ks	25. july. 2011	rev 1.2
	HEAD Informationen geändert, neuer Spaltenzähler

ks	16. apr. 2012	rev 1.3
	neuer überarbeiteter Code für automatisches File-open/close

ks	8. mar. 2016	rev 1.4
	nur einmal nach satellitenbausteinen scannen

ks	21. mar. 2016	rev 1.5
	prüfung auf freien bufferplatz hinzugefügt
	fehlermeldungen hinzugefügt
*)

END_FUNCTION_BLOCK

// POUs/DEMO/DLOG_FILE_CSV_FTP_DEMO
PROGRAM DLOG_FILE_CSV_FTP_DEMO
VAR
	cur_dt: DT;
	enable: BOOL := TRUE;
	trig_t : TIME := T#5s;
	trig_m : BOOL;
	error_c: DWORD;
	error_t: BYTE;
	auto_close: TIME := T#10s;

	x1: DLOG_DT;
	x2 : DLOG_REAL;
	x3 : DLOG_DINT;
	x4 : DLOG_BOOL;
	x5: DLOG_STRING;
	x : DLOG_DATA;
	RTC_2: oscat_basic.RTC_2;
	DLOG_STORE_FILE_CSV : DLOG_STORE_FILE_CSV;
	GEN_SIN_1: oscat_basic.GEN_SIN;
	COUNT_DR: oscat_basic.COUNT_DR;

	DLOG_FILE_TO_FTP: DLOG_FILE_TO_FTP;
	ftp_done: BOOL;
	ftp_busy: BOOL;
	ftp_error_c: DWORD;
	ftp_error_t: BYTE;
	ftp_url: STRING := 'ftp://581920:123456@oscat.atwebpages.com:2000/subordner/';
	ftp_activ: BOOL := FALSE;
	ftp_delete: BOOL := TRUE;
	ftp_retry: INT := 0;
	ftp_retry_time: TIME := T#60s;
	ftp_timeout: TIME := T#30s;
END_VAR

VAR RETAIN
	save_data : DLOG_SAVE;
END_VAR
VAR // added by the converter: edge detectors and wires of the graphical bodies
    _w1, _w2, _w3 : ANY;
END_VAR

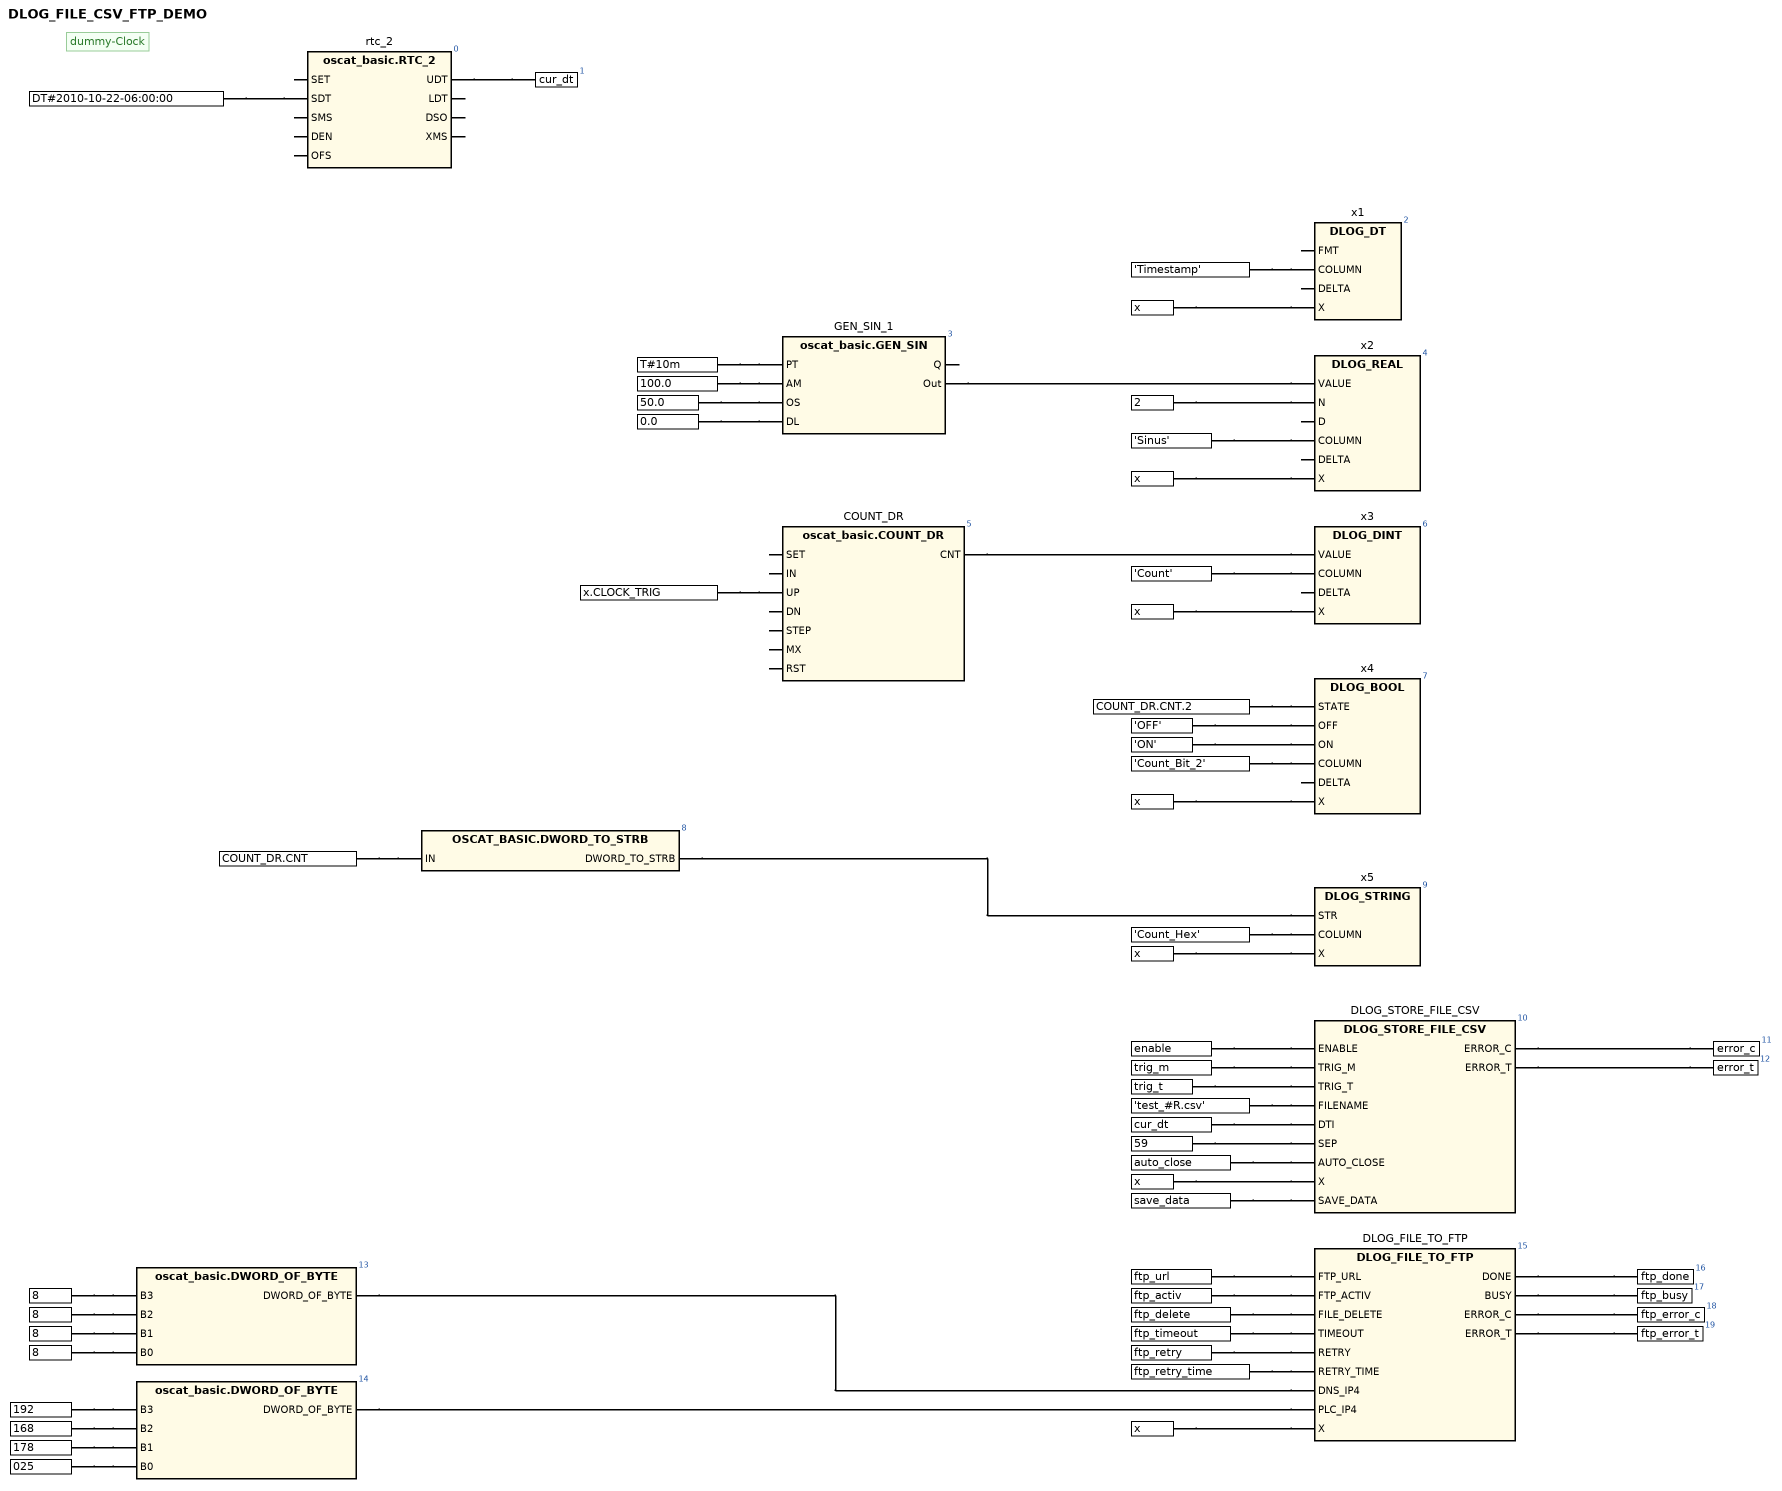
// dummy-Clock
rtc_2(SDT := DT#2010-10-22-06:00:00); // oscat_basic.RTC_2
cur_dt := rtc_2.UDT;
x1(COLUMN := 'Timestamp', X := x); // DLOG_DT
GEN_SIN_1(PT := T#10m, AM := 100.0, OS := 50.0, DL := 0.0); // oscat_basic.GEN_SIN
x2(VALUE := GEN_SIN_1.Out, N := 2, COLUMN := 'Sinus', X := x); // DLOG_REAL
COUNT_DR(UP := x.CLOCK_TRIG); // oscat_basic.COUNT_DR
x3(VALUE := COUNT_DR.CNT, COLUMN := 'Count', X := x); // DLOG_DINT
x4(STATE := COUNT_DR.CNT.2, OFF := 'OFF', ON := 'ON', COLUMN := 'Count_Bit_2', X := x); // DLOG_BOOL
_w1 := OSCAT_BASIC.DWORD_TO_STRB(IN := COUNT_DR.CNT);
x5(STR := _w1, COLUMN := 'Count_Hex', X := x); // DLOG_STRING
DLOG_STORE_FILE_CSV(
    ENABLE := enable,
    TRIG_M := trig_m,
    TRIG_T := trig_t,
    FILENAME := 'test_#R.csv',
    DTI := cur_dt,
    SEP := 59,
    AUTO_CLOSE := auto_close,
    X := x,
    SAVE_DATA := save_data);
error_c := DLOG_STORE_FILE_CSV.ERROR_C;
error_t := DLOG_STORE_FILE_CSV.ERROR_T;
_w2 := oscat_basic.DWORD_OF_BYTE(B3 := 8, B2 := 8, B1 := 8, B0 := 8);
_w3 := oscat_basic.DWORD_OF_BYTE(B3 := 192, B2 := 168, B1 := 178, B0 := 025);
DLOG_FILE_TO_FTP(
    FTP_URL := ftp_url,
    FTP_ACTIV := ftp_activ,
    FILE_DELETE := ftp_delete,
    TIMEOUT := ftp_timeout,
    RETRY := ftp_retry,
    RETRY_TIME := ftp_retry_time,
    DNS_IP4 := _w2,
    PLC_IP4 := _w3,
    X := x);
ftp_done := DLOG_FILE_TO_FTP.DONE;
ftp_busy := DLOG_FILE_TO_FTP.BUSY;
ftp_error_c := DLOG_FILE_TO_FTP.ERROR_C;
ftp_error_t := DLOG_FILE_TO_FTP.ERROR_T;

END_PROGRAM

// POUs/DATA_LOG/DLOG_FILE_TO_FTP
FUNCTION_BLOCK DLOG_FILE_TO_FTP
VAR_IN_OUT
	X : DLOG_DATA;
END_VAR
VAR_INPUT
	FTP_URL : STRING(OSCAT_BASIC.STRING_LENGTH);
	FTP_ACTIV : BOOL;
	FILE_DELETE : BOOL;
	TIMEOUT : TIME := T#30s;
	RETRY : INT;
	RETRY_TIME : TIME := T#30s;
	DNS_IP4 : DWORD;
	PLC_IP4 : DWORD;
END_VAR
VAR_OUTPUT
	DONE : BOOL;
	BUSY : BOOL;
	ERROR_C : DWORD;
	ERROR_T : BYTE;
END_VAR
VAR
	UCBD : UNI_CIRCULAR_BUFFER_DATA;
	UCB : UNI_CIRCULAR_BUFFER;
	FTP_CLIENT : FTP_CLIENT;
	WT_1 : TON;
	ftrig_old : BOOL;
	filename : STRING;
	step : INT;
	ftp_busy : BOOL;
	ftp_done : BOOL;
	cnt : INT;

	(*LOG_MSG : LOG_MSG;
	_debug_enable : BOOL := TRUE;*)
END_VAR

(*
version 1.2		21. mar. 2016
programmer		ks
tested by			ks

DLOG_FILE_TO_FTP der Baustein kopiert bzw verschiebt die vom DLOG_STORE_FILE_CSV erzeugten Dateien auf einem FTP-Server
*)

(* neue Filenamen speichern *)
IF X.NEW_FILE_RTRIG AND ftrig_old = FALSE THEN
	UCBD.D_HEAD := 1;
	UCBD.D_MODE := 1;
	UCBD.D_STRING := X.NEW_FILE;
	UCB(DATA:=UCBD); (* Daten eintragen *)
END_IF;
ftrig_old := X.NEW_FILE_RTRIG;

CASE step OF

00:	IF UCBD.BUF_COUNT > 0 AND ftp_busy = FALSE THEN
		UCBD.D_MODE := 12; (* Daten lesen und löschen *)
		UCB(DATA:=UCBD);
		filename := UCBD.D_STRING;
		cnt := RETRY;
		step := 10;

		(*####################  DEBUG-MESSAGE  ###################################*)
		(*IF _debug_enable THEN
			LOG_CL.NEW_MSG := 'F_T_FTP: Auftrag aktiv /file: ~2';
			LOG_CL.PRINTF[2] := files;
			LOG_MSG();
		END_IF;*)
		(*########################################################################*)

	END_IF;

10:	IF ftp_busy = FALSE THEN
		IF ftp_done THEN
			(*####################  DEBUG-MESSAGE  ###################################*)
			(*IF _debug_enable THEN
				LOG_CL.NEW_MSG := 'F_T_FTP: Auftrag OK /file: ~2';
				LOG_CL.PRINTF[2] := filename;
				LOG_MSG();
			END_IF;*)
			(*########################################################################*)
			step := 0;
		ELSE
			step := 20; (* pause nach error *)
		END_IF;
	END_IF;

20:	IF WT_1.Q THEN (* Wartezeit *)
		cnt := cnt - 1;
		IF RETRY = 0 THEN (* FTP Transfer unbegrenzt wiederholen *)
			(*####################  DEBUG-MESSAGE  ###################################*)
			(*IF _debug_enable THEN
				LOG_CL.NEW_MSG := 'F_T_FTP: Auftrag unbegrenzt wiederholen /file: ~2';
				LOG_CL.PRINTF[2] := filename;
				LOG_MSG();
			END_IF;*)
			(*########################################################################*)
			step := 10; (* FTP Transfer wiederholen *)
		ELSIF cnt >= 0 THEN
			(*####################  DEBUG-MESSAGE  ###################################*)
			(*IF _debug_enable THEN
				LOG_CL.NEW_MSG := 'F_T_FTP: Auftrag wiederholen /cnt: ~1 /file: ~2';
				LOG_CL.PRINTF[1] := INT_TO_STRING(cnt);
				LOG_CL.PRINTF[2] := filename;
				LOG_MSG();
			END_IF;*)
			(*########################################################################*)
			step := 10; (* FTP Transfer wiederholen *)
		ELSE
			(*####################  DEBUG-MESSAGE  ###################################*)
			(*IF _debug_enable THEN
				LOG_CL.NEW_MSG := 'F_T_FTP: Auftrag verworfen /file: ~2';
				LOG_CL.PRINTF[2] := filename;
				LOG_MSG();
			END_IF;*)
			(*########################################################################*)
			step := 0; (* FTP Auftrag verwerfen *)
		END_IF;
	END_IF;

END_CASE;

BUSY := step = 10;
DONE := step = 0;
WT_1(IN:= step = 20, PT:= RETRY_TIME);

FTP_CLIENT(
	ACTIVATE:= BUSY,
	FILENAME:= filename,
	FTP_URL:= FTP_URL,
	FTP_DOWNLOAD:= FALSE,
	FTP_ACTIV:= FTP_ACTIV,
	FILE_DELETE:= FILE_DELETE,
	TIMEOUT:= TIMEOUT,
	DNS_IP4:= DNS_IP4,
	PLC_IP4:= PLC_IP4,
	DONE=> ftp_done,
	BUSY=> ftp_busy
	);

(* Fehlerauswertung *)
IF FTP_CLIENT.ERROR_T <> BYTE#0 THEN
	ERROR_C := FTP_CLIENT.ERROR_C;
	ERROR_T := FTP_CLIENT.ERROR_T;
ELSIF UCBD.BUF_DATA_LOST > UDINT#0 THEN
	ERROR_C := DWORD#2; (* Fehler: Bufferüberlauf - Datenmenge reduzieren *)
	ERROR_T := BYTE#6; 	(* Type: Buffer *)
ELSIF UCBD.BUF_USED_MAX > USINT#90 THEN
	ERROR_C := DWORD#1; (* Warnung: Buffer auslastung > 90% *)
	ERROR_T := BYTE#6;	(* Type: Buffer *)
ELSE
	ERROR_C := DWORD#0;
	ERROR_T := BYTE#0;
END_IF;

(* revision history
ks	01. jan. 2011	rev 1.0
	original version

ks	26. jul. 2011	rev 1.1
    codeoptimierung D_MODE 12

ks	21. mar. 2016	rev 1.2
	fehlermeldungen hinzugefügt
	fehler in RETRY korrigiert
	
*)

END_FUNCTION_BLOCK

// POUs/NETWORK/FTP_CLIENT
FUNCTION_BLOCK FTP_CLIENT
VAR_INPUT
	ACTIVATE : BOOL;
	FILENAME : STRING;
	FTP_URL : STRING(OSCAT_BASIC.STRING_LENGTH);
	FTP_DOWNLOAD : BOOL;
	FTP_ACTIV : BOOL;
	FILE_DELETE : BOOL;
	TIMEOUT : TIME;
	DNS_IP4 : DWORD;
	PLC_IP4 : DWORD;
END_VAR
VAR_OUTPUT
	DONE : BOOL;
	BUSY : BOOL;
	ERROR_C : DWORD;
	ERROR_T : BYTE;
END_VAR
VAR
	IP_C1 : IP_C; (* IP_Control Verwaltungsstruktur *)
	IP_C2 : IP_C; (* IP_Control Verwaltungsstruktur *)
	S_BUF1 : NETWORK_BUFFER;
	S_BUF2 : NETWORK_BUFFER;
	R_BUF1 : NETWORK_BUFFER;
	R_BUF2 : NETWORK_BUFFER;
	URL_DATA : url;
	DNS_CLIENT : DNS_CLIENT;
	IPC1 : IP_CONTROL;
	IPC2 : IP_CONTROL;
	FS : FILE_SERVER;
	FSD : FILE_SERVER_DATA;

	activate_last : BOOL;
	step : INT;
	snd_step : INT;
	snd_text :	STRING(OSCAT_BASIC.STRING_LENGTH);
	rcv_text :	STRING(OSCAT_BASIC.STRING_LENGTH);
	rcv_state : INT;
	TON_WAIT : TON;
	last_step : INT;
	next_step : INT;
	idx1 : INT;
	idx2 : INT;
	str1 : STRING(OSCAT_BASIC.STRING_LENGTH);
	str2 : STRING(OSCAT_BASIC.STRING_LENGTH);
	ftp_path : STRING;
	byar : ARRAY [0..5] OF BYTE;
	dw_tmp : DWORD;
	w_tmp : WORD;
	fpd : FILE_PATH_DATA;
	timeout2 : TIME;
	timeout3 : TIME;
	ftp_file_size : UDINT;
	ip_c1_red_disable : BOOL; (* IP_CONTROL 1 - Remote Disconnect Error unterdrücken *)
	ip_c2_red_disable : BOOL; (* IP_CONTROL 1 - Remote Disconnect Error unterdrücken *)

	(*LOG_MSG : LOG_MSG;
	_debug_enable : BOOL := FALSE;*)

END_VAR
(*
version 1.3		05.may 2012
programmer		ks
tested by			ks

FTP_CLIENT dient zum senden und empfangen von dateien von einem FTP-Server.



110 Restart marker reply 										Markierung für Wiederaufnahme der Übertragung 
120 Service ready in x minutes 									Dienst steht in x Minuten zu Verfügung 
125 Data connection already open; 								transfer starting Datenverbindung besteht bereits; beginne mit der Übertragung 
150 File status okay; about to open data connection 					Dateistatus OK; Datenverbindung wird aufgebaut 
200 Command okay 											Befehl OK 
202 Command not implemented 									Befehl nicht implementiert 
211   														Antwort für Systemstatus oder Hilfefunktion des Systems 
212   														Verzeichnisstatus 
213   														Dateistatus 
214   														Meldung der Hilfefunktion 
215 NAME system type 										Angabe des Systemtyps 
220 Service ready for new user 									Dienst bereit für neuen Benutzer 
221 Service closing control connection 							Steuerverbindung des Dienstes wird getrennt; Benutzer wird abgemeldet 
225 Data connection open; no transfer in progress 					Datenverbindung hergestellt; derzeit keine Übertragung 
226 Closing data connection. Requested file action successful 		Datenverbindung wird getrennt 
227 Entering Passive Mode 										Passiver Modus aktiviert 
230 User logged in, proceed 									Benutzer angemeldet, bitte fortfahren 
250 Requested file action okay, completed 						Angeforderter Vorgang OK, beendet 
257 "PATH" created 											"PFAD" wurde erstellt 
331 User name okay, need password 							Benutzername OK, Kennwort erforderlich 
332 Need account for login 										Benutzerkonto zur Anmeldung erforderlich 
350 Requested file action pending further information 				Mehr Informationen für Dateivorgang erforderlich 
421 Service not available, closing control connection 				Dienst nicht verfügbar, Steuerverbindung wird getrennt 
425 Can't open data connection 									Datenverbindung kann nicht hergestellt werden 
426 Connection closed; transfer aborted Verbindung getrennt; 		Übertragung abgebrochen 
450 Requested file action not taken; File unavailable 				Angeforderter Dateivorgang wurde nicht ausgeführt; Datei nicht verfügbar 
451 Requested action aborted: local error in processing 				Angeforderter Vorgang abgebrochen: Lokaler Fehler bei der Bearbeitung 
452 Requested action not taken; Insufficient storage space in system 	Angeforderter Vorgang nicht ausgeführt; Nicht genügend Speicherplatz auf System 
500 Syntax error 												Befehl nicht erkannt 
501 Syntax error in parameters or arguments 						Syntaxfehler bei den Parametern 
502 Command not implemented 									Befehl nicht implementiert 
503 Bad sequence of commands 								Ungültige Befehlsabfolge 
504 Command not implemented for that parameter 					Befehl für diesen Parameter nicht implementiert 
530 Not logged in 												Nicht angemeldet 
532 Need account for storing files 								Zum Speichern von Dateien Anmeldung erforderlich 
550 Requested file action not taken; File unavailable Angeforderter 	Dateivorgang wurde nicht ausgeführt; Datei nicht verfügbar 
551 Requested action aborted: page type unknown 					Angeforderter Vorgang abgebrochen: Unbekannter Seitentyp 
552 Requested file action aborted: Exceeded storage allocation 		Angeforderter Dateivorgang abgebrochen: Nicht genügend Platz in aktuellem Verzeichnis oder Datensatz 
553 Requested action not taken: File name not allowed 				Angeforderter Vorgang nicht ausgeführt: Unzulässiger Dateiname 

#########################
ERROR_T

1 = DNS_CLIENT
2 = FTP Steuerkanal
3 = FTP Datenkanal
4 = FILE_SERVER
5 = Ablaufstörung
#########################

*)

CASE step OF

00:	IF ACTIVATE AND NOT activate_last THEN
		ftp_file_size := UDINT#0;
		TIMEOUT := MAX(T#10s,TIMEOUT);
		timeout2 := TIMEOUT + T#1s;
		timeout3 := TIMEOUT / 2;
		DONE := FALSE;
		ip_c1_red_disable := FALSE;
		ip_c2_red_disable := FALSE;
		ERROR_C := DWORD#0;
		ERROR_T := BYTE#0;
		FSD.ERROR := BYTE#0;
		URL_DATA := STRING_TO_URL(STR:=FTP_URL,DEFAULT_PROTOCOL:='',DEFAULT_PATH:='/');
		IF LEN(URL_DATA.USER) = 0 THEN
			URL_DATA.USER := 'Anonymous';
			URL_DATA.PASSWORD := 'User@';
		END_IF;

		FILE_PATH_SPLIT(FILENAME:=FILENAME,X:=fpd); (* Datei-Path zerlegen *)
		str1 := fpd.FILENAME; (* zwischenspeichern *)
		FILE_PATH_SPLIT(FILENAME:=URL_DATA.PATH,X:=fpd); (* FTP-Path zerlegen *)
		IF LEN(fpd.FILENAME) = 0 THEN (* wenn FTP-Path keinen Dateinamen enthält , dann den Namen der lokalen Datei benutzen *)
			ftp_path := CONCAT(URL_DATA.PATH,str1);
		ELSE
			ftp_path := URL_DATA.PATH;
		END_IF;
		step := 10;
	END_IF;

10:	IF DNS_CLIENT.DONE THEN
		step := 20;
	ELSIF DNS_CLIENT.ERROR <> DWORD#0 THEN
		ERROR_C := DNS_CLIENT.ERROR;
		ERROR_T := BYTE#1;
		step := 980;
	END_IF;

20:	(* FTP Steuerkanal einrichten *)
	IP_C1.C_PORT := WORD#21; (* Portnummer eintragen *)
  	IP_C1.C_IP := DNS_CLIENT.IP4; (* IP eintragen *)
  	IP_C1.C_MODE := BYTE#0; (* Mode: TCP+ACTIV+PORT *)
  	IP_C1.TIME_RESET := TRUE; (* Zeitueberwachung rücksetzen *)
  	IP_C1.C_ENABLE := TRUE; (* Verbindungsaufbau freigeben *)
  	IP_C1.R_OBSERVE := TRUE; (* Empfangsueberwachung *)
	R_BUF1.SIZE := UINT#0;

  	IP_C2.C_ENABLE   := FALSE; (* Verbindungsaufbau sperren *)
	step := 30;

30:	IF rcv_state = 220 THEN (* 220 = Service ready for new user *)
		snd_text := CONCAT('USER ',URL_DATA.USER);
		next_step := 40;
	END_IF;

40:	IF rcv_state = 331 THEN (* 331 = User name okay, need password *)
		snd_text := CONCAT('PASS ',URL_DATA.PASSWORD);
		next_step := 50;
	ELSIF rcv_state = 230 THEN (* 230 = User logged in, proceed *)
		next_step := 50;
	ELSIF rcv_state = 220 THEN (* 220 = Service ready for new user *)
		next_step := 20; (* WORK verbindung sollte ab/aufgebaut werden *)
	END_IF;

50:	IF rcv_state = 230 THEN (* 230 = User logged in, proceed *)
		snd_text := 'TYPE I';  (* binären Modus aktivieren *)
		next_step := 54;
	END_IF;

54:	IF rcv_state = 200 THEN (* 200 = Command okay *)
		IF FTP_DOWNLOAD THEN (* Datei von FTP Empfangen *)
			snd_text := CONCAT('SIZE ', ftp_path); (* SIZE /PFAD/FILENAME *)
			next_step := 56;
		ELSE
			step := 60;
		END_IF;
	END_IF;

56:	IF rcv_state = 213 THEN (* 213 Filesize *)
		str1 := ELEMENT_GET(SEP:=BYTE#32,POS:=1,ELEMENT:=rcv_text);
		ftp_file_size := STRING_TO_UDINT(str1); (* Dateigroesse in bytes gestimmen *)
		step := 60;
	END_IF;

60:	IF FTP_ACTIV THEN (* FTP Server aktiv *)
		IF URL_DATA.PORT = WORD#0 THEN
			URL_DATA.PORT := WORD#20; (* Standard Datenkanal *)
		END_IF;
		str2 := '';
		dw_tmp := PLC_IP4;
		FOR idx1 := 0 TO 5 DO
			IF idx1 = 4 THEN
				dw_tmp := ROR(WORD_TO_DWORD(URL_DATA.PORT),8);
			ELSE
				dw_tmp := ROL(dw_tmp,8);
			END_IF;
			str2 := CONCAT(str2,BYTE_TO_STRING(DWORD_TO_BYTE(dw_tmp)));
			IF idx1 < 5 THEN
				str2 := CONCAT(str2,',');
			END_IF;
		END_FOR;
		dw_tmp := DNS_CLIENT.IP4; (* IP eintragen *)
		w_tmp := URL_DATA.PORT; (* Port Nummer des Datenkanals *)
		snd_text := CONCAT('PORT ',str2); (* FTP Server in den aktiv-mode schalten *)
		next_step := 80;
	ELSE
		snd_text := 'PASV';  (* FTP Server in den passiv-mode schalten *)
		next_step := 70;
	END_IF;
	step := 999; (* Warten auf next_step *)

70:	IF rcv_state = 227 THEN (* 227 = Entered Passive Mode (213,202,225,43,212,186) *)
		idx1 := FIND(rcv_text , '(' );
		idx2 := FIND(rcv_text , ')' );
		IF idx1 > 0 AND idx2 > idx1+1 THEN
			str1 := MID(rcv_text, idx2 - idx1 - 1, idx1+1);
			FOR idx1 := 0 TO 5 DO
				str2 := ELEMENT_GET(SEP:=BYTE#44,POS:=idx1,ELEMENT:=str1);
				byar[idx1] := STRING_TO_BYTE(str2);
			END_FOR;
			dw_tmp := OSCAT_BASIC.DWORD_OF_BYTE(byar[0],byar[1],byar[2],byar[3]); (* IP Adresse des Datenkanals *)
			w_tmp := OSCAT_BASIC.WORD_OF_BYTE(byar[4],byar[5]); (* Port Nummer des Datenkanals *)
		END_IF;
		step := 100;
	END_IF;

80:	IF rcv_state = 200 THEN (* 200 = PORT command successful *)
		step := 100;
	END_IF;

100:IP_C2.C_MODE := SEL(FTP_ACTIV,BYTE#0,BYTE#2); (* Aktiv = Mode 2: TCP+PASSIV+PORT / passiv = Mode 0: TCP+ACTIV+PORT *)
	IP_C2.C_IP := dw_tmp; (* IP Adresse des Datenkanals *)
	IP_C2.C_PORT := w_tmp; (* Port Nummer des Datenkanals *)
  	IP_C2.TIME_RESET := TRUE; (* Zeitueberwachung rücksetzen *)
  	IP_C2.C_ENABLE := TRUE; (* Verbindungsaufbau freigeben *)
	IP_C2.R_OBSERVE := FALSE; (* Empfangsueberwachung *)
	R_BUF2.SIZE := UINT#0;
	step := 120;

120:IF IP_C2.C_STATE > BYTE#127 THEN (* FTP Datenkanal aufgebaut *)
		IF FTP_DOWNLOAD THEN (* File von FTP empfangen *)
			IP_C2.MAILBOX[3] := BYTE#1; (* IP Empfang sperren *)
			step := 400;
		ELSE
			snd_text := 'STOR ';
			next_step := 140;
			snd_text := CONCAT(snd_text, ftp_path); (* STORE /PFAD/FILENAME *)
			step := 999; (* Warten auf next_step *)
		END_IF;
	END_IF;

(* ============== File an FTP senden ================ *)

140:IF rcv_state = 125 OR rcv_state = 150 THEN (* 125 = Data connection already open / 150 = File status okay; about to open data connection *)
		step := 160;
	END_IF;

160:FSD.FILENAME := FILENAME; (* Dateiname *)
	FSD.MODE := BYTE#1; (* vorhandene Datei zum lesen öffnen *)
	FSD.OFFSET := UDINT#0; (* Start bei Dateianfang *)
	S_BUF2.SIZE := UINT#65535; (* maximale länge einlesen *)
	IP_C2.MAILBOX[2] := BYTE#1; (* IP Senden blockieren *)
	step := 200;

200:IF FSD.MODE = BYTE#0 AND FSD.ERROR = BYTE#0 THEN
		IP_C2.MAILBOX[2] := BYTE#0; (* IP Senden erlauben *)
		step := 210;
	END_IF;

210:IF S_BUF2.SIZE = UINT#0 THEN (* warten bis alle daten gesendet sind *)
		IF FSD.FILE_SIZE - FSD.OFFSET > UDINT#0 THEN
			FSD.MODE := BYTE#1; (* vorhandene Datei zum lesen öffnen *)
			S_BUF2.SIZE := UINT#65535; (* maximale länge einlesen *)
			IP_C2.MAILBOX[2] := BYTE#1; (* IP Senden blockieren *)
			step := 200;
		ELSE
			IP_C2.C_ENABLE := FALSE; (* FTP Datenkanal schliessen *)
			step := 300;
		END_IF;
	END_IF;

300:IF rcv_state = 226 THEN (* 226 Closing data connection. Requested file action successful  *)
		snd_text := 'QUIT';
		ip_c1_red_disable := TRUE;
		next_step := 320;
	END_IF;

320:IF rcv_state = 221 OR TON_WAIT.ET > timeout3  THEN (* 221 Service closing control connection *)
		IP_C1.C_ENABLE := FALSE; (* FTP Steuerkanal schliessen *)
		IF FILE_DELETE THEN (* Datei nach transfer löschen *)
			FSD.MODE := BYTE#4; (* File Remove *)
			step := 340;
		ELSE
			step := 900;
		END_IF;
	END_IF;

340:IF FSD.MODE = BYTE#0 AND FSD.ERROR = BYTE#0 THEN
		step := 900;
	END_IF;

(*  ============== File vom FTP Empfangen  ============== *)

400:snd_text := 'RETR ';
	next_step := 410;
	snd_text := CONCAT(snd_text, ftp_path); (* RETR /PFAD/FILENAME *)
	step := 999; (* Warten auf next_step *)

410:IF rcv_state = 125 OR rcv_state = 150 THEN (* 125 = Data connection already open / 150 = File status okay; about to open data connection *)
		IP_C2.R_OBSERVE := TRUE; (* Empfangsueberwachung *)
		step := 420;
	END_IF;

420:FSD.FILENAME := FILENAME; (* Dateiname *)
	FSD.MODE := BYTE#3; (* Datei neu anlegen *)
	FSD.OFFSET := UDINT#0; (* Start bei Dateianfang *)
	step := 460;

440:IF R_BUF2.SIZE > UINT#0 THEN (* warten bis daten empfangen wurden *)
		IP_C2.MAILBOX[3] := BYTE#1; (* IP Empfang blockieren bis Daten in Datei geschrieben wurden *)
		FSD.MODE := BYTE#3; (* Daten in Datei schreiben *)
		step := 460;
	ELSIF FSD.FILE_SIZE = ftp_file_size THEN (* Verbindung abgebaut ? , oder 226 = Closing data connection. Requested file action successful *)
		IP_C2.C_ENABLE := FALSE; (* FTP Datenkanal schliessen *)
		ip_c2_red_disable := TRUE;
		step := 700;
	END_IF;

460:IF FSD.MODE = BYTE#0 AND FSD.ERROR = BYTE#0 THEN (* warten bis Daten geschreiben wurden *)
		R_BUF2.SIZE := UINT#0; (* Daten löschen *)
		IP_C2.MAILBOX[3] := BYTE#0; (* IP Empfang wieder erlauben *)
		step := 440;
	END_IF;

(* ================================================== *)

700:IF rcv_state = 226 OR  TON_WAIT.ET > timeout3 THEN (* 226 Closing control connection. Requested file action successful  *)
		IF FTP_DOWNLOAD AND FILE_DELETE THEN (* FTP Download und File löschen ? *)
			snd_text := CONCAT('DELE ', ftp_path); (* DELE /PFAD/FILENAME *)
			next_step := 720;
		ELSE
			step := 740;
		END_IF;
	END_IF;

720:IF rcv_state = 250 THEN (* 250 Requested file action okay, completed *)
		step := 740;
	END_IF;

740:snd_text := 'QUIT';
	ip_c1_red_disable := TRUE;
	next_step := 760;
	step := 999; (* Warten auf next_step *)

760:IF rcv_state = 221 OR TON_WAIT.ET > timeout3 THEN (* 221 Service closing control connection  *)
		IP_C1.C_ENABLE := FALSE; (* FTP Steuerkanal schliessen *)
		IF NOT FTP_DOWNLOAD AND FILE_DELETE THEN (* FTP Upload und Datei nach transfer löschen *)
			FSD.MODE := BYTE#4; (* File Remove *)
			step := 780;
		ELSE
			step := 900;
		END_IF;
	END_IF;

780:IF FSD.MODE = BYTE#0 AND FSD.ERROR = BYTE#0 THEN
		step := 900;
	END_IF;

(* ================================================== *)

900:DONE := TRUE;
	step := 980;

980:IP_C1.C_ENABLE := FALSE; (* FTP Steuerkanal schliessen *)
	IP_C2.C_ENABLE := FALSE; (* FTP Datenkanal schliessen *)
	IP_C2.MAILBOX[2] := BYTE#0; (* IP Senden wieder erlauben *)
	IP_C2.MAILBOX[3] := BYTE#0; (* IP Empfang wieder erlauben *)
	S_BUF1.SIZE := UINT#0;
	S_BUF2.SIZE := UINT#0;
	R_BUF1.SIZE := UINT#0;
	R_BUF2.SIZE := UINT#0;
	ftp_file_size := UDINT#0;
	snd_step := 0;
	next_step := 0;
	FSD.MODE := BYTE#5; (* Datei schliessen *)
	step := 990;

990:IF IP_C1.C_STATE = BYTE#0 AND IP_C2.C_STATE = BYTE#0 AND FSD.FILE_OPEN = FALSE THEN
		step := 0;
	END_IF;

999: ; (* Dummy Schritt, warten bis neuer schritt durch "next_step" aktiv wird *)

END_CASE;

(* ++++++++++++++++++++++++++++++++++++++++++++++++++++++++++ *)

IF step >= 30 THEN
	IF R_BUF1.SIZE > UINT#0 THEN (* Daten wurden empfangen ? *)
		idx1 := UINT_TO_INT(R_BUF1.SIZE);
		REPEAT (* zeilenterminierung erkennen und echtes TEXT-Ende bestimmen *)
			idx1 := idx1 - 1;
		UNTIL idx1 = 0 OR R_BUF1.BUFFER[idx1] >= BYTE#32 (* TRUE = EXIT *)
		END_REPEAT;
		idx1 := idx1 + 1; (* index auf SIZE umrechnen *)
		rcv_text := OSCAT_BASIC.BUFFER_TO_STRING(PT:=ADR(R_BUF1.BUFFER),SIZE:=idx1,START:=0,STOP:=OSCAT_BASIC.STRING_LENGTH-1);
		IF LEN(rcv_text) >= 3 THEN (* Statuscode prüfen und auswerten *)
			str1 := LEFT(rcv_text,3);
			IF OSCAT_BASIC.IS_NUM(STR:=str1) THEN (* enthält nur Zahlen ? *)
				rcv_state := STRING_TO_INT(str1);
			END_IF;
			IP_C1.R_OBSERVE := FALSE;
		END_IF;
		R_BUF1.SIZE := UINT#0; (* daten löschen *)

	        (*####################  DEBUG-MESSAGE  ###################################*)
	        (*IF _debug_enable THEN
	          LOG_CL.NEW_MSG := 'RCV: >~1<';
	          LOG_CL.PRINTF[1] := rcv_text;
	          LOG_MSG();
	        END_IF;*)
	        (*########################################################################*)

	END_IF;
END_IF;

(* automatisches Datensenden *)

CASE snd_step OF

00:	IF LEN(snd_text) > 0 THEN
	        (*####################  DEBUG-MESSAGE  ###################################*)
	        (*IF _debug_enable THEN
	          LOG_CL.NEW_MSG := 'SND: >~1<';
	          LOG_CL.PRINTF[1] := snd_text;
	          LOG_MSG();
	        END_IF;*)
	        (*########################################################################*)
		OSCAT_BASIC._STRING_TO_BUFFER(str:=snd_text,pos:=0,pt:=ADR(S_BUF1.BUFFER),size:=SIZEOF(S_BUF1.BUFFER)); (* String in puffer kopieren *)
		idx1 := LEN(snd_text);
		S_BUF1.BUFFER[idx1] := BYTE#16#0D;
		idx1 := idx1 + 1;
		S_BUF1.BUFFER[idx1] := BYTE#16#0A;
		idx1 := idx1 + 1;
		S_BUF1.SIZE := INT_TO_UINT(idx1); (* Sendelänge eintragen *)
		R_BUF1.SIZE := UINT#0; (* Empfangsbuffer rücksetzen *)
		IP_C1.R_OBSERVE := TRUE;
		rcv_state := 9999; (* letzen FTP Status löschen *)
		snd_text := '';
		snd_step := 10;
	END_IF;

10:	IF S_BUF1.SIZE = UINT#0 THEN (* warten bis alle daten gesendet sind *)
		step := next_step;
		snd_step := 0;
	END_IF;

END_CASE;

(* Globale Fehlerbehandlung für Haupt-Routine *)
IF ERROR_T = BYTE#0 AND step > 20 THEN (* noch kein Fehler gespeichert und Hauptroutine aktiv *)

	IF IP_C1.ERROR > DWORD#0 AND IP_C1.C_ENABLE AND NOT IP_C1.TIME_RESET THEN  (* IP Control 1 *)
		IF ip_c1_red_disable = FALSE OR IP_C1.ERROR <> DWORD#16#FD000000 THEN
			ERROR_C := IP_C1.ERROR;
			ERROR_T := BYTE#2;
			step := 980;
		END_IF;
	END_IF;

	IF IP_C2.ERROR > DWORD#0 AND IP_C2.C_ENABLE AND NOT IP_C2.TIME_RESET THEN  (* IP Control 2 *)
		IF ip_c2_red_disable = FALSE OR IP_C2.ERROR <> DWORD#16#FD000000 THEN
			ERROR_C := IP_C2.ERROR;
			ERROR_T := BYTE#3;
			step := 980;
		END_IF;
	END_IF;

	IF FSD.MODE = BYTE#0 THEN
		IF FSD.ERROR > BYTE#0 THEN
			ERROR_C := BYTE_TO_DWORD(FSD.ERROR);
			ERROR_T := BYTE#4; (* Dateizugriff *)
			step := 980;
		END_IF;
	END_IF;
END_IF;

IF TON_WAIT.Q THEN (* Ablaufstörung - Schrittkette *)
	ERROR_C := SHL(INT_TO_DWORD(step),16) OR INT_TO_DWORD(rcv_state); (* aktuellen Schritt und letzten FTP Status eintragen *)
	ERROR_T := BYTE#5;
	step := 980;
END_IF;

(* ######################################################## *)

DNS_CLIENT(IP_C:=IP_C1, S_BUF:=S_BUF1, R_BUF:=R_BUF1, DOMAIN:=URL_DATA.DOMAIN, IP4_DNS:= DNS_IP4, ACTIVATE:=step=10); (* DNS-Client *)
IPC1(IP:= DWORD#0, PORT:= WORD#0 , TIME_OUT:= TIMEOUT, IP_C:= IP_C1, S_BUF:= S_BUF1, R_BUF:= R_BUF1); (* FTP Steuerkanal *)
IPC2(IP:= DWORD#0, PORT:= WORD#0 , TIME_OUT:= TIMEOUT, IP_C:= IP_C2, S_BUF:= S_BUF2, R_BUF:= R_BUF2); (* FTP Datenkanal *)

TON_WAIT(IN:=step = last_step AND step > 0,PT:=timeout2);
last_step := step;
activate_last := ACTIVATE;
BUSY := step <> 0;

IF FTP_DOWNLOAD THEN (* FILE_SERVER *)
	FS(FSD:=FSD,PT:=R_BUF2); (* Datei von FTP empfangen *)
ELSE
	FS(FSD:=FSD,PT:=S_BUF2); (* Datei an FTP senden *)
END_IF;

(* revision history
ks	05. may 2011	rev 1.3
	FileServer AutoClose entfernt

ks	11. may 2011	rev 1.2
	ip_control - remote disconnect error ausblenden, und sonderbehandlung für pcworx

ks	06. apr. 2011	rev 1.1
	list_len und list_get durch element_count und element_get ersetzt

ks	01. jan. 2011	rev 1.0
	original version
*)

END_FUNCTION_BLOCK

// POUs/CONVERT/STRING_TO_URL
FUNCTION STRING_TO_URL : URL
VAR_INPUT
	STR : STRING(OSCAT_BASIC.STRING_LENGTH);
	DEFAULT_PROTOCOL : STRING(10);
	DEFAULT_PATH : STRING(80);
END_VAR
VAR
	pos: INT;
	pos2: INT;
	x : STRING(OSCAT_BASIC.STRING_LENGTH);
END_VAR

(*
version 1.3	04. mar. 2016
programmer 	hugo
tested by		oscat

URL splits a unifrom resource locator in its conponents.

*)

(*

http://hans:geheim@www.example.org:80/demo/example.cgi?land=de&stadt=aa#abschnitt1
|       |      |         |         |   |                   |               |
|       |      |         Host      |   Pfad                Query           Anker
|       |      Passwort            Port
|       Benutzer
Protokoll

*)

(* check if string is empty and return empty url *)
IF STR = '' THEN RETURN; END_IF;

(* extract the protocol *)
(* first we check if the optional protocol is specified ending with a :// *)
pos := FIND(STR, '://');
IF pos > 0 THEN
	(* store protocol and restore the rest of url in temp *)
	STRING_TO_URL.PROTOCOL := LEFT(STR, pos - 1);
	x := RIGHT(STR, LEN(STR) - pos - 2);
ELSE
	x := STR;
	STRING_TO_URL.PROTOCOL := DEFAULT_PROTOCOL;
END_IF;

(* extract user and password if present ending with a @ *)
pos := OSCAT_BASIC.FINDB(STR1:=x,STR2:='@'); (* Find last @ *)

IF pos > 0 THEN
	(* extract user *)
	pos2 := FIND(x,':')+1;
	IF pos2 > 1 AND pos2 <= pos THEN
		STRING_TO_URL.USER := LEFT(x,pos2 - 2);
		STRING_TO_URL.PASSWORD := MID(x, pos - pos2, pos2);
	ELSE
		STRING_TO_URL.USER := LEFT(x, pos - 2);
		STRING_TO_URL.PASSWORD := '';
	END_IF;
	x := RIGHT(x, LEN(x) - pos);
ELSE
	STRING_TO_URL.USER := '';
	STRING_TO_URL.PASSWORD := '';
END_IF;

(* extract anchor *)
pos := FIND(x, '#');
IF pos > 0 THEN
	STRING_TO_URL.ANCHOR := RIGHT(x, LEN(x) - pos);
	x := LEFT(x, pos - 1);
ELSE
	STRING_TO_URL.ANCHOR := '';
END_IF;

(* extract query  *)
pos := FIND(x, '?');
IF pos > 0 THEN
	STRING_TO_URL.QUERY := RIGHT(x, LEN(x) - pos);
	x := LEFT(x, pos - 1);
ELSE
	STRING_TO_URL.QUERY := '';
END_IF;

(* extract path  *)
pos := FIND(x, '/');
IF pos > 0 THEN
	STRING_TO_URL.PATH := RIGHT(x, LEN(x) - pos + 1);
	x := LEFT(x, pos - 1);
ELSE
	STRING_TO_URL.PATH := DEFAULT_PATH;
END_IF;

(* extract port and leave domain *)
pos := FIND(x, ':');
IF pos > 0 THEN
	STRING_TO_URL.PORT := STRING_TO_WORD(RIGHT(x, LEN(x) - pos));
	STRING_TO_URL.DOMAIN := LEFT(x, pos - 1);
ELSE
	STRING_TO_URL.PORT := 0;
	STRING_TO_URL.DOMAIN := x;
END_IF;

(* revision history
hm		18. apr 2008	rev 1.0
	original version

ks		20. dec. 2010	rev 1.1
	stringlength 250 , var x

ks		27. oct. 2012	rev 1.2
	var_temp zu var geändert

ks		04. mar. 2016	rev 1.3
	@ zeichen wird nun von rechts nach links gesucht
	ermöglicht username und password mit @ zeichen
*)

END_FUNCTION

// POUs/FILE/FILE_PATH_SPLIT
FUNCTION FILE_PATH_SPLIT : BOOL
VAR_INPUT
	FILENAME : STRING(OSCAT_BASIC.STRING_LENGTH);
END_VAR
VAR_IN_OUT
	X : FILE_PATH_DATA;
END_VAR
VAR
	b : INT;
	c : INT;
	d : STRING(1);
	p1 : INT;
	p2 : INT;
END_VAR

(*
version 1.0		01. jan. 2011
programmer		ks
tested by			ks

FILE_PATH_SPLIT zerlegt einen Dateipfad in einzelne Elemente und legt diese in einer Datenstruktur ab.
*)

X.DRIVE := '';
X.DIRECTORY := '';
X.FILENAME := '';
c := LEN(FILENAME);
IF c = 0 THEN
	FILE_PATH_SPLIT := FALSE;
	RETURN;
END_IF;

FOR b := 1 TO c DO
	d := MID(FILENAME, 1, b);
	IF d = ':' THEN
		p1 := b;
	ELSIF d = '/' OR d = '\' THEN
		p2 := b;
	END_IF;
END_FOR;

IF p1 = 2 THEN
	X.DRIVE := LEFT(FILENAME,p1);
END_IF;

IF p2 > 0 AND p2 > p1 THEN
	X.DIRECTORY := MID(FILENAME,p2 - p1,p1+1); (* len , pos *)
END_IF;

X.FILENAME := RIGHT(FILENAME,c - MAX (p1,p2));
FILE_PATH_SPLIT := TRUE;

(* revision history
ks	01. jan. 2011	rev 1.0
	original version
*)

END_FUNCTION

// POUs/NETWORK/DNS_CLIENT
FUNCTION_BLOCK DNS_CLIENT
VAR_IN_OUT
	IP_C : IP_C; (* IP_Control Verwaltungsstruktur *)
	S_BUF : NETWORK_BUFFER;
	R_BUF : NETWORK_BUFFER;
END_VAR
VAR_INPUT
	ACTIVATE : BOOL;
	DOMAIN : STRING;
	IP4_DNS : DWORD;
END_VAR
VAR_OUTPUT
	IP4 : DWORD;
	DONE : BOOL;
	ERROR : DWORD;
END_VAR
VAR
	IP_FIFO : IP_FIFO;
	ip_state : BYTE;
	ip_id : BYTE;
	i : INT;
	state : INT;
	domain_copy : STRING;
	activate_last : BOOL;
	url_length : INT;
	char : BYTE;
	char_count : INT;
	tid : BYTE;
	anc : INT;
	x : BYTE;
	rr_stop : BOOL;
	ttl_last : DWORD;
	ttl_tmp : DWORD;

	(*LOG_MSG : LOG_MSG;
	_debug_enable : BOOL := TRUE;*)

END_VAR

(*
version 1.3	26. jul. 2011
programmer 	ks
tested BY	ks

DNS_CLIENT führt eine Domain-Name Abfrage bei einen DNS-Server durch

*)

(* Domain Name System (query) *)

CASE state OF

00:	IF ACTIVATE AND NOT activate_last THEN (* auf positive Flanke GET warten *)
		DONE := FALSE;
		ERROR := DWORD#0;
		state := 5;
	END_IF;

05:	IP4 := IP4_DECODE(str:=DOMAIN); (* prüfe ob domain schon eine IP4-Adresse ist *)
	IF IP4 > DWORD#00 THEN
		DONE := TRUE;
		state := 0;
        		(*####################  DEBUG-MESSAGE  ###################################*)
        		(*IF _debug_enable THEN
            		LOG_CL.NEW_MSG := 'DNS: S05 IP4 ~1';
            		LOG_CL.PRINTF[1]  := DOMAIN;
            		LOG_MSG();
        		END_IF;*)
        		(*########################################################################*)
	ELSE
		ip_state := BYTE#1;
		ttl_last := DWORD#0;
		domain_copy := DOMAIN; (* DOMAIN String sichern *)
		state := 10;
        		(*####################  DEBUG-MESSAGE  ###################################*)
        		(*IF _debug_enable THEN
            		LOG_CL.NEW_MSG := 'DNS: S05 START';
            		LOG_MSG();
        		END_IF;*)
        		(*########################################################################*)
	END_IF;

10:	IF ip_state = BYTE#3 THEN (* Bei IP_Control anmelden *)
		url_length := LEN(domain_copy);
		char_count := 17 + url_length; (* sendebuffer initialisieren *)
		FOR i := 0 TO char_count DO
			S_BUF.BUFFER[i] := BYTE#00;
		END_FOR;
		tid := UINT_TO_BYTE(BYTE_TO_UINT(tid) + UINT#1);
		S_BUF.BUFFER[01] := tid; (* Transaction ID lowbyte *)
		S_BUF.BUFFER[02] := BYTE#16#01; (* Flags: highbyte *)
		S_BUF.BUFFER[05] := BYTE#16#01; (* Questions: lowbyte *)
		i := url_length + 12;	(* den servernamen von hinten nach vorne bearbeiten *)
		char_count := 0;
		WHILE i > 12 DO
			char := OSCAT_BASIC.CODE(STR:=domain_copy,POS:=i - 12);
			IF char = BYTE#46 THEN (* prüfe auf haupt/sub domänen namens-teiler "." *)
				S_BUF.BUFFER[i] := INT_TO_BYTE(char_count); (* anstelle des teilers "." wird die länge des erkannten haupt/sub domänennames eingetragen *)
				char_count := 0;
			ELSE
				S_BUF.BUFFER[i] := char; (* char in buffer eintragen *)
				char_count := char_count + 1; (* anzahl char zählen *)
			END_IF;
			i := i - 1;
		END_WHILE;
		S_BUF.BUFFER[i] := INT_TO_BYTE(char_count); (* längenangabe des ganz linken (ersten) domänennamens eintragen *)
		i := url_length + 15; (* position hinter dem servernamen *)
		S_BUF.BUFFER[i] := BYTE#01; (* Type: A Hostaddress lowbyte *)
		i := i + 2;
		S_BUF.BUFFER[i] := BYTE#01; (* Class: IN lowbyte *)
		i := i + 1;
		(* IP Datenverkehr einrichten *)
		IP_C.C_PORT := WORD#53; (* Portnummer eintragen *)
		IP_C.C_IP := IP4_DNS; (* IP eintragen *)
		IP_C.C_MODE := BYTE#1; (* Mode: UDP+AKTIV+PORT+IP *)
		IP_C.C_ENABLE := TRUE; (* Verbindungsaufbau freigeben *)
		IP_C.TIME_RESET := TRUE; (* Zeitueberwachung rücksetzen *)
		IP_C.R_OBSERVE  := TRUE; (* Datenempfang ueberwachen *)
		S_BUF.SIZE := INT_TO_UINT(i); (* sendelänge eintragen *)
		R_BUF.SIZE := UINT#0; (* Empfangslänge rücksetzen *)
		state := 30;

        		(*####################  DEBUG-MESSAGE  ###################################*)
        		(*IF _debug_enable THEN
            		LOG_CL.NEW_MSG := 'DNS: S10 SEND';
            		LOG_MSG();
        		END_IF;*)
        		(*########################################################################*)
	END_IF;

30:	IF IP_C.ERROR <> DWORD#00 THEN
		ERROR := IP_C.ERROR;
		state := 99;
        		(*####################  DEBUG-MESSAGE  ###################################*)
        		(*IF _debug_enable THEN
            		LOG_CL.NEW_MSG := 'DNS: S30 ERROR ~1';
            		LOG_CL.PRINTF[1]  := DWORD_TO_STRING(ERROR);
            		LOG_MSG();
        		END_IF;*)
        		(*########################################################################*)

	ELSIF (S_BUF.SIZE = UINT#0) AND (tid = R_BUF.BUFFER[1]) AND (R_BUF.SIZE >= INT_TO_UINT(34 + url_length)) THEN	(* prüfe ob antwort telegramm die richtige Transaction-ID und mindestlänge hat *)
		ERROR := BYTE_TO_DWORD(R_BUF.BUFFER[3] AND BYTE#2#0000_1111); (* prüfe Return code der Flags. 4 bits *)
		IF ERROR = DWORD#00 THEN
			anc := R_BUF.BUFFER[7]; (* Anzahl der Answer-RR *)
			IP_C.R_OBSERVE := FALSE; (* Datenempfang ueberwachen *)
			state := 40;
		ELSE
			state := 99;
		END_IF;
	END_IF;

40:	IF anc > 0 THEN
		anc := anc - 1;
		WHILE i < R_BUF.SIZE DO
			x := R_BUF.BUFFER[i];
			IF rr_stop = FALSE THEN
				IF x > BYTE#63 THEN (* zeiger auf namen *)
					i := i + 1;
					rr_stop := TRUE;
				ELSIF x= BYTE#0 THEN (* namens ende *)
					rr_stop := TRUE;
				ELSE
					i := i + x; (* namen *)
				END_IF;
				i := i + 1;
			ELSE
				rr_stop := FALSE;
				IF R_BUF.BUFFER[i+1] = BYTE#1 AND R_BUF.BUFFER[i+3] = BYTE#1 THEN (* Type A / Class IN *)
					i := i + 4;
					ttl_tmp := OSCAT_BASIC.DWORD_OF_BYTE(R_BUF.BUFFER[i],R_BUF.BUFFER[i+1],R_BUF.BUFFER[i+2],R_BUF.BUFFER[i+3]); (* Time to live *)
					i := i + 6;
					IF ttl_tmp >= ttl_last THEN (* TTL ist länger *)
						ttl_last := ttl_tmp;
						IP4 := OSCAT_BASIC.DWORD_OF_BYTE(R_BUF.BUFFER[i],R_BUF.BUFFER[i+1],R_BUF.BUFFER[i+2],R_BUF.BUFFER[i+3]); (* IP-Adresse *)
					END_IF;
					i := i + 4;
				ELSE
					i := i + 9;
					i := i + R_BUF.BUFFER[i] + 1; (* offset zu nächsten Block *)
				END_IF;
				EXIT;
			END_IF;
		END_WHILE;
	ELSE
		IF IP4 > DWORD#0 THEN (* gültige RR mit IP gefunden *)
			DONE := TRUE;
            		(*####################  DEBUG-MESSAGE  ###################################*)
            		(*IF _debug_enable THEN
                			LOG_CL.NEW_MSG := 'DNS: S40 OK';
                			LOG_MSG();
            		END_IF;*)
            		(*########################################################################*)
		ELSE
			ERROR := DWORD#255; (* Daten fehlerhaft - keine IP-Adresse vorhanden *)
		END_IF;
		state := 99;
	END_IF;

99:	R_BUF.SIZE := UINT#0; (* Empfangslänge rücksetzen *)
	ip_state := BYTE#4; (* Abmelden *)
	state := 00;

END_CASE;

activate_last := ACTIVATE; (* letzten Status sichern zur Flankenerkennung *)
IP_FIFO(FIFO:=IP_C.FIFO,STATE:=ip_state,ID:=ip_id); (* IP_FIFO *)

(* revision history

ks	18. oct. 2008	rev 1.0
	original version

ks	20. oct. 2009	rev 1.1
	unbenutzten code entfernt, all buffer base 0

ks	20. dec. 2010	rev 1.2
	parsing nach rfc1305

ks	26. jul. 2011	rev 1.3
	verbesserte ip-auswertung , neue fehlermeldung
*)


(*----------------------------------------------------------------------------------------------------------------*)
(* Flags: 0x0100 (Standard query)                                                                                            *)
(* 0... .... .... .... = Response: Message is a query                                                                   *)
(* .000 0... ....  = Opcode: Standard query (0)                                                                          *)
(* .... ..0. .... .... = Truncated: Message is not truncated                                                          *)
(* .... ...1 .... .... = Recursion desired: Do query recursively                                                    *)
(* .... .... .0.. .... = Z: reserved (0)                                                                                                  *)
(* .... .... ...0 .... = Non-authenticated data OK: Non-authenticated data is unacceptable *)
(*-----------------------------------------------------------------------------------------------------------------*)

(*      0  1  2  3  4  5  6  7  8  9  0  1  2  3  4  5  *)
(*    +--+--+--+--+--+--+--+--+--+--+--+--+--+--+--+--+ *)
(*    |                      ID                       | idx: 0/1   *)
(*    +--+--+--+--+--+--+--+--+--+--+--+--+--+--+--+--+ *)
(*    |QR|   Opcode  |AA|TC|RD|RA|   Z    |   RCODE   | idx: 2/3   *)
(*    +--+--+--+--+--+--+--+--+--+--+--+--+--+--+--+--+ *)
(*    |                    QDCOUNT                    | idx: 4/5   *)
(*    +--+--+--+--+--+--+--+--+--+--+--+--+--+--+--+--+ *)
(*    |                    ANCOUNT                    | idx: 6/7   *)
(*    +--+--+--+--+--+--+--+--+--+--+--+--+--+--+--+--+ *)
(*    |                    NSCOUNT                    | idx: 8/9   *)
(*    +--+--+--+--+--+--+--+--+--+--+--+--+--+--+--+--+ *)
(*    |                    ARCOUNT                    | idx: 10/11 *)
(*    +--+--+--+--+--+--+--+--+--+--+--+--+--+--+--+--+ *)

(*
Errorcodes  Description	References 
000	No error. 		 	The request completed successfully.
001	Format error. 		The name server was unable to interpret the query. 
002	Server failure.  	The name server was unable to process this query due to a problem with the name server. 
003	Name Error. 	 	Meaningful only for responses from an authoritative name server, this code signifies that the domain name referenced in the query does not exist.
004	Not Implemented. 	The name server does not support the requested kind of query.
005	Refused. 			The name server refuses to perform the specified operation for policy reasons.
  						 For example, a name server may not wish to provide the information to the particular requester, or a name server may not wish to perform a particular operation (e.g., zone transfer) for particular data.
006	YXDomain.			Name Exists when it should not. 
007	YXRRSet. RR			Set Exists when it should not. 
008	NXRRSet. RR			Set that should exist does not. 
009	NotAuth.			Server Not Authoritative for zone. 
010	NotZone,			Name not contained in zone. 
255	Timeout				No Response  
   

beispiel einer DNS Request von google.at
ein request mit 3 Answer-Blocks


Domain Name System (response)
[Request In: 3]
[Time: 0.027533000 seconds]
Transaction ID: 0x5e1a
Flags: 0x8180 (Standard query response, No error)
1... .... .... .... = Response: Message is a response
.000 0... .... .... = Opcode: Standard query (0)
.... .0.. .... .... = Authoritative: Server is not an authority for domain
.... ..0. .... .... = Truncated: Message is not truncated
.... ...1 .... .... = Recursion desired: Do query recursively
.... .... 1... .... = Recursion available: Server can do recursive queries
.... .... .0.. .... = Z: reserved (0)
.... .... ..0. .... = Answer authenticated: Answer/authority portion was not authenticated
.... .... .... 0000 = Reply code: No error (0)
Questions: 1
Answer RRs: 3
Authority RRs: 0
Additional RRs: 0

Queries
google.at: type A, class IN
Name: google.at
Type: A (Host address)
Class: IN (0x0001)

Answers
google.at: type A, class IN, addr 72.14.221.104
Name: google.at
Type: A (Host address)
Class: IN (0x0001)
Time to live: 19 minutes, 9 seconds
Data length: 4
Addr: 72.14.221.104

google.at: type A, class IN, addr 66.249.93.104
Name: google.at
Type: A (Host address)
Class: IN (0x0001)
Time to live: 19 minutes, 9 seconds
Data length: 4
Addr: 66.249.93.104

google.at: type A, class IN, addr 216.239.59.104
Name: google.at
Type: A (Host address)
Class: IN (0x0001)
Time to live: 19 minutes, 9 seconds
Data length: 4
Addr: 216.239.59.104
*)

END_FUNCTION_BLOCK

// POUs/CONVERT/IP4_DECODE
FUNCTION IP4_DECODE : DWORD
VAR_INPUT
	str : STRING(15);
END_VAR
VAR
	pos: INT;
END_VAR

(*
version 1.1	10. mar 2009
programmer 	kurt
tested by		hugo

IP4_DECODE testet ob ein string eine gültige IPv4 Adresse enthält und gibt die 4 Bytes der IP Adresse als DWORD zurück.

*)

pos := FIND(str, '.');
WHILE pos > 0 DO
	IP4_DECODE := SHL(IP4_DECODE,8) OR STRING_TO_DWORD(LEFT(str,pos - 1));
	str := DELETE(str, pos, 1);
	pos := FIND(str, '.');
END_WHILE;
IP4_DECODE := SHL(IP4_DECODE,8) OR STRING_TO_DWORD(str);


(* revision history
hm		29. feb 2008	rev 1.0
	original version

hm	10. mar. 2009	rev 1.1
	new algorythm
*)

END_FUNCTION

// POUs/HARDWARE/IP_CONTROL
FUNCTION_BLOCK IP_CONTROL
VAR_IN_OUT
	IP_C : IP_C; (* IP_Control Verwaltungsstruktur *)
	S_BUF : NETWORK_BUFFER; (* Externer Sendbuffer *)
	R_BUF : NETWORK_BUFFER; (* Externer Receivebuffer *)
END_VAR
VAR_INPUT
	IP : DWORD; (* IP Adresse *)
	PORT : WORD; (* Port Nummer *)
	TIME_OUT : TIME; (* Ueberwachungszeit Connect / Send / Receive *)
END_VAR
VAR
	c_time : UDINT; (* CONNECT-Time (Zeit bei nicht vorhandener Verbindung) *)
	s_time : UDINT; (* SEND-Time    (Zeit seit letzten Datensenden) *)
	r_time : UDINT; (* RECEIVE-Time (Zeit seit letztem Datenempfang) *)

	c_enable : BOOL; (* Connect: freigabe *)
	c_ip : DWORD; (* Connect: aktuelle IP-Adresse *)
	c_port : WORD; (* Connect: aktuelle Port-Nummer *)
	c_mode : BYTE; (* Connect: aktueller Mode UDP/TCP...... *)
	c_status : BYTE; (* Connect: Status (Errorcode) *)
	c_ready : BOOL; (* Connect: Verbindung aufgebaut *)
	c_ready_old : BOOL; (* Connect: letzter Zustand von c_ready für Flankenauswertung *)
	c_select : BOOL; (* non blocking mode - abfrage über select durchführen *)
	c_fdWrite : SOCKET_FD_SET;
	c_Timeout : SOCKET_TIMEVAL;

	s_total : INT; (* Send: Gesamtanzahl Bytes zum senden *)
	s_cur_pos : INT; (* Send: aktuelle Sendeposition *)
	s_cur_size : INT; (* Send: aktuelle Sendegroesse *)
	s_max_size : INT; (* Send: maximale Telegrammlänge fuer Senden *)
	s_start : BOOL; (* Send: Sende modus aktivieren *)
	s_active : BOOL; (* Send: Daten senden ist aktiv *)
	s_req : BOOL; (* Send: Start Daten senden *)
	s_done : BOOL; (* Send: ohne Fehler beendet *)
	s_status : BYTE; (* Send: Status (Errorcodes) *)

	r_status : BYTE; (* Receive: Status (Errorcodes) *)
	r_count : INT; (* Receive: Anzahl empfangener Bytes *)
	r_offset : INT; (* Receive: aktuelle Position in externen Receivebuffer *)
	r_max_size : INT; (* Receive: groesse des externen Empfangbuffers*)

	new_connection : BOOL; (* Neue Verbindungsparameter vorhanden *)
	tx : DWORD; (* letzter zeitwert *)
	error_time : DWORD; (* aktueller Timeout-Wert *)

	state: BYTE; (* schrittmerker für connect *)
	server_socket : DINT:= SOCKET_INVALID;
	socket : DINT:= SOCKET_INVALID;
	sockaddr : SOCKADDRESS;
	sockaddr_size : DWORD;
	plc_841 : BOOL;
	plc_881 : BOOL;
	dint_true : DINT := 1;
	bytes_received : DINT;
	bytes_sent : DINT;
	udp_mode : BOOL;

	(*LOG_MSG : LOG_MSG;
	_debug_enable : BOOL := TRUE;
	debug_index : INT;
	debug_ID : INT;
	debug_lasterror : DWORD;
	debug_last_id : INT := 255;
	state_last: BYTE;*)

END_VAR

VAR CONSTANT
	STOP : BYTE := 0;
	TS_INIT: BYTE := 1;
	TS_OPEN : BYTE:= 2;

	UDP_INIT : BYTE:= 31;

	TC_INIT : BYTE:= 51;
	TC_CONNECT : BYTE:= 52;

	C_WAIT : BYTE:= 250;
	C_CLOSE : BYTE:= 251;

END_VAR

(*

version 1.9		26. Feb. 2012
programmer 		ks
tested by			ks

IP_CONTROL ist ein Wrapper-Baustein um eine Hersteller neutrale Schnittstelle zum Ethernet zu schaffen
*)

(* ---------------------- Debug-Message ----------------------------*)
(*IF _debug_enable THEN
	IF IP_C.FIFO.ID > BYTE#0 THEN
		debug_index := IP_C.FIFO.NR;
		debug_ID := BYTE_TO_INT(IP_C.FIFO.X[debug_index]);
	END_IF;
END_IF;*)
(* -----------------------------------------------------------------------------*)

(* read system time *)
tx := OSCAT_BASIC.T_PLC_MS();

IF IP_C.C_PORT = 0 THEN
	IP_C.C_PORT := PORT; (* uebergebenen PORT durch parametrierten PORT ersetzen *)
END_IF;
IF IP_C.C_IP = 0 AND IP_C.C_MODE < 4 THEN
	IP_C.C_IP := IP; (* uebergebene IP durch paramtrierte IP ersetzen *)
END_IF;

new_connection := c_ip <> IP_C.C_IP OR c_mode <> IP_C.C_MODE OR c_port <> IP_C.C_PORT; (* neue Verbindungs erwünscht ? *)
c_enable := IP_C.C_ENABLE AND NOT new_connection;

IF IP_C.C_ENABLE AND IP_C.ERROR = 0 AND state = STOP THEN (* Freigabe,kein Fehler,kein Socket offen *)
	c_ip   := IP_C.C_IP;
	c_mode := IP_C.C_MODE;
	c_port := IP_C.C_PORT;
	plc_841 := SYSLIBSOCKETS_OPTION.1; (* Bit 1 = WAGO 750-841 *)
	plc_881 := SYSLIBSOCKETS_OPTION.2; (* Bit 1 = WAGO 750-881 *)
	udp_mode := C_MODE.0; (* Mode 1,3,5 = udp *)

	error_time := TIME_TO_DWORD(MAX(T#200ms,TIME_OUT));
	IP_C.TIME_RESET := TRUE; (* Alle Timer ruecksetzen *)

	r_max_size := SIZEOF(R_BUF.BUFFER);
	s_max_size := SIZEOF(S_BUF.BUFFER);

	IF C_MODE.0 THEN (* Mode: 1,3,5 = UDP CLIENT/SERVER *)
		state := UDP_INIT;
	ELSIF C_MODE = 0 THEN (* Mode: 0 = TCP CLIENT *)
		state := TC_INIT;
	ELSE
		state := TS_INIT; (* Mode: 2,4 = TCP SERVER *)
	END_IF;

	(* ---------------------- Debug-Message ----------------------------*)
	(*IF _debug_enable THEN
		LOG_CL.NEW_MSG := 'IP_CON: MODE ~1 / IP ~2 / PORT ~3 /ID ~6';
		LOG_CL.PRINTF[1] := BYTE_TO_STRING(C_MODE);
		LOG_CL.PRINTF[2] := IP4_TO_STRING(c_ip);
		LOG_CL.PRINTF[3] := WORD_TO_STRING(c_port);
		LOG_CL.PRINTF[6] := INT_TO_STRING(debug_ID);
		LOG_MSG();
	END_IF;*)
	(* -----------------------------------------------------------------------------*)

END_IF;

(* ---------------------- Debug-Message ----------------------------*)
(*IF  _debug_enable THEN
	IF state <> state_last THEN
		LOG_CL.NEW_MSG := 'IP_STEP ~1 -IP_ID ~6';
		LOG_CL.PRINTF[1] := BYTE_TO_STRING(state);
		LOG_CL.PRINTF[6] := INT_TO_STRING(debug_ID);
		LOG_MSG();
		state_last := state;
	END_IF;
END_IF;*)
(* -----------------------------------------------------------------------------*)

IF IP_C.TIME_RESET THEN (* Alle Timer ruecksetzen *)
	IP_C.TIME_RESET := FALSE; (* Reset rücksetzen *)
	c_time := tx; (* Connect Timer ruecksetzen *)
	s_time := tx; (* Send Timer ruecksetzen *)
	r_time := tx; (* Receive Timer ruecksetzen *)

	c_status := BYTE#0; (* letzten Connect Fehler rücksetzen *)
	s_status := BYTE#0; (* letzten Send Fehler rücksetzen *)
	r_status := BYTE#0; (* letzten Receive Fehler rücksetzen *)
END_IF;

(* ---------------------------------------------- *)

CASE state OF

UDP_INIT: (* UDP_CLIENT + SERVER *)
	socket := SysSockCreate(SOCKET_AF_INET, SOCKET_DGRAM, SOCKET_IPPROTO_IP);
	IF socket < 0 THEN
		c_status := 1; (* SysSockCreate failed *)
		state := C_CLOSE;
	ELSE
		SysSockSetOption(socket, SOCKET_SOL, SOCKET_SO_BROADCAST, ADR(dint_true), SIZEOF(dint_true)); (* allow broadcast *)
		SysSockIoctl(socket, SOCKET_FIONBIO, ADR(dint_true)); (* put socket in non-blocking mode *)
		sockaddr.sin_family := SOCKET_AF_INET;
		sockaddr.sin_port := SysSockHtons(c_port);
		sockaddr.sin_addr := SEL(c_mode = 1, SOCKET_INADDR_ANY, SysSockNtohl(c_ip));

		IF c_mode >= 2 THEN (* SERVER Mode *)
			IF SysSockBind(socket, ADR(sockaddr), SIZEOF(sockaddr)) THEN
				c_ready := TRUE; (* Connected *)
				state:= C_WAIT;
			ELSE
				c_status := 2; (* SysSockBind failed *)
				state := C_CLOSE;
			END_IF;
		ELSE
			c_ready := TRUE; (* Connected *)
			state:= C_WAIT;
		END_IF;
	END_IF;

(* ---------------------------------------------- *)

TC_INIT: (* TCP-CLIENT (AKTIV) *)
	socket := SysSockCreate(SOCKET_AF_INET, SOCKET_STREAM, SOCKET_IPPROTO_IP);
	IF socket < 0 THEN
		c_status := 1;  (* SysSockCreate failed *)
		state := C_CLOSE;
	ELSE
		IF plc_841 OR plc_881 THEN
			SysSockSetOption(socket,6,SOCKET_TCP_NODELAY, ADR(dint_true), SIZEOF(dint_true)); (* Set Push-Bit *)
		END_IF;
		SysSockIoctl(socket, SOCKET_FIONBIO, ADR(dint_true)); (* NonBlocking mode *)
		sockaddr.sin_family := SOCKET_AF_INET;
		sockaddr.sin_port := SysSockNtohs(c_port);
		sockaddr.sin_addr := SysSockNtohl(c_ip);
		c_select := FALSE;
		state := TC_CONNECT;
	END_IF;

(* ---------------------------------------------- *)

TC_CONNECT:
	IF NOT c_enable OR c_status = 255 THEN (* keine freigabe oder connect timeout *)
			state:= C_CLOSE;
	ELSE
		IF c_select = FALSE THEN
			IF SysSockConnect(socket,ADR(sockaddr),SIZEOF(sockaddr)) THEN
				c_ready := TRUE; (* Connected *)
				state:= C_WAIT;
			ELSE
				(* Connect durchgeführt, aber noch nicht verbunden, dann optional mit select-abfrage weitermachen *)
				c_select := SYSLIBSOCKETS_OPTION.0; (* Bit 0 = TCP-Client - use SysSockselect *)
			END_IF;
		ELSE
			c_Timeout.tv_sec := 0;
			c_Timeout.tv_usec := 0;
			c_fdWrite.fd_count := 1;
			c_fdWrite.fd_array[0] := socket;
			IF SysSockSelect(SOCKET_FD_SETSIZE,0,ADR(c_fdWrite),0, ADR(c_Timeout)) > 0 THEN
				c_ready := TRUE; (* Connected *)
				state:= C_WAIT;
			END_IF;
		END_IF;
	END_IF;

(* ---------------------------------------------- *)

TS_INIT: (* TCP-SERVER (PASSIV) *)
	server_socket := SysSockCreate(SOCKET_AF_INET, SOCKET_STREAM, SOCKET_IPPROTO_IP); (* Create Socket *)
	IF server_socket = SOCKET_INVALID THEN
		c_status := 1; (* SysSockCreate failed *)
		state:= C_CLOSE;
	ELSE (* Address bindings *)
		SysSockSetOption( server_socket, SOCKET_SOL, SOCKET_SO_REUSEADDR, ADR(dint_true), SIZEOF(dint_true) );
		sockaddr.sin_family:= SOCKET_AF_INET;
		sockaddr.sin_port := SysSockHtons(c_port);
		sockaddr.sin_addr := SOCKET_INADDR_ANY;
		IF NOT SysSockBind(server_socket, ADR(sockaddr), SIZEOF(sockaddr)) THEN
			c_status := 2; (* SysSockBind failed *)
			state := C_CLOSE;
		ELSIF NOT SysSockListen(server_socket, 1) THEN (* erzeugt Warteschlange für eine Verbindung *)
			c_status := 3; (* SysSockListen failed *)
			state:= C_CLOSE;
		ELSE
			SysSockIoctl(server_socket, SOCKET_FIONBIO, ADR(dint_true)); (* NonBlocking mode *)
			state:= TS_OPEN;
		END_IF;
	END_IF;

(* ---------------------------------------------- *)

TS_OPEN: (* Waiting for incomming connection *)
	sockaddr_size := SIZEOF(sockaddr);
	socket := SysSockAccept(server_socket, ADR(sockaddr), ADR(sockaddr_size));

	IF socket <> SOCKET_INVALID THEN (* neuer Verbindungswunsch vorhanden *)
		IF c_mode = BYTE#2 AND sockaddr.sin_addr <> SysSockNtohl(c_ip) THEN (* Mode 2 = TCP + PASSIVE + PORT + IP  auf richtige Partner-IP prüfen *)
			state:= C_CLOSE;
		ELSE
			IF plc_841 OR plc_881 THEN
				SysSockSetOption(socket, 6, SOCKET_TCP_NODELAY, ADR(dint_true), SIZEOF(dint_true)); (* Set Push-Bit *)
			END_IF;
			SysSockIoctl(socket, SOCKET_FIONBIO, ADR(dint_true)); (* NonBlocking mode *)
			c_ready := TRUE; (* Connected *)
			state := C_WAIT;
		END_IF;
	ELSIF NOT c_enable THEN (* keine freigabe mehr ? *)
			state:= C_CLOSE;
	END_IF;

(* ---------------------------------------------- *)

C_WAIT: (* Warten auf Anforderung für Beenden *)
	IF NOT c_enable OR NOT c_ready THEN
		state:= C_CLOSE;
	END_IF

(* ---------------------------------------------- *)

C_CLOSE: (* Close the Sockets *)
	c_ready := FALSE;
	IF socket >= 0 THEN
		IF (NOT plc_841) AND (NOT plc_881) THEN
			SysSockShutdown(socket, 0); (* 870 *)
		END_IF;
		SysSockClose(socket);
		socket := SOCKET_INVALID;
	END_IF
	IF server_socket >= 0 THEN
		IF (NOT plc_841) AND (NOT plc_881) THEN
			SysSockShutdown(server_socket, 0); (* 870 *)
		END_IF;
		SysSockClose(server_socket);
		server_socket := SOCKET_INVALID;
	END_IF
	state:= STOP;
END_CASE;

(* ---------------------------------------------- *)

IF c_ready THEN
	IF NOT c_ready_old THEN (* Verbindung aufgebaut - positive Flanke erkannt *)
		IP_C.C_STATE := 254;
		IP_C.TIME_RESET := TRUE; (* Alle Timer ruecksetzen *)
		(* ---------------------- Debug-Message ----------------------------*)
		(*IF _debug_enable THEN
			LOG_CL.NEW_MSG := 'IP_CON: CONNECTED -IP_ID ~6';
			LOG_CL.PRINTF[6] := INT_TO_STRING(debug_ID);
			LOG_MSG();
		END_IF;*)
		(* -----------------------------------------------------------------------------*)
	ELSE
		IP_C.C_STATE := 255; (* Verbindung ist aufgebaut *)
	END_IF;
ELSE
	IF c_ready_old THEN (* Verbindung abgebaut - negative Flanke erkannt *)
		IP_C.C_STATE := 1;
		IP_C.MAILBOX[1] := 0; (* Receive Info rücksetzen *)
		IP_C.MAILBOX[2] := 0; (* Send-Pause rücksetzen *)
		IP_C.MAILBOX[3] := 0; (* Receive-Pause rücksetzen *)
		IF NOT new_connection THEN
			s_active := FALSE; (* Sendeaktivitäten stoppen *)
			s_req := FALSE; (* Sendefreigabe rücksetzen *)
			S_BUF.SIZE := 0; (* Sendelänge löschen *)
			(*IP_C.TIME_RESET := TRUE;*) (* Alle Timer ruecksetzen *)
		END_IF;
		(* ---------------------- Debug-Message ----------------------------*)
		(*IF _debug_enable THEN
			LOG_CL.NEW_MSG := 'IP_CON: DISCONNECTED';
			LOG_MSG();
		END_IF;*)
		(* -----------------------------------------------------------------------------*)
	ELSE
		IP_C.C_STATE := 0; (* Verbindung ist abgebaut *)
	END_IF;
END_IF;

c_ready_old := c_ready;

(* Der Datenempfang wird angehalten solange ein Sendevorgang läuft *)
(* sonst kann es vorkommen das die Antwort-daten schon empfangen werden, *)
(* bevor der Sendevorgang vom programm abgeschlossen wurde *)

IF c_ready AND NOT s_active AND IP_C.MAILBOX[3] = 0 THEN
	IF R_BUF.SIZE >= INT_TO_UINT(r_max_size) THEN
		R_BUF.SIZE := UINT#0;
		r_status := 254; (* Empfangsbuffer wegen Überlauf rückgesetzt *)
	END_IF;

	r_offset := SEL(udp_mode,UINT_TO_INT(R_BUF.SIZE),0);
	r_count := r_max_size - r_offset;

	IF udp_mode THEN
		bytes_received := SysSockRecvFrom(socket, ADR(R_BUF.BUFFER), r_count, 0, ADR(sockaddr), SIZEOF(sockaddr));

		IF c_mode = BYTE#3 AND sockaddr.sin_addr <> SysSockNtohl(c_ip) THEN (* Mode 3 = UDP + PASSIVE + PORT + IP  auf richtige Partner-IP prüfen *)
			bytes_received := 0;
			R_BUF.SIZE := UINT#0;
			sockaddr.sin_port := SysSockNtohs(c_port);
			sockaddr.sin_addr := SysSockNtohl(c_ip);
		END_IF;

	ELSE
		bytes_received := SysSockRecv(socket, ADR(R_BUF.BUFFER[r_offset]), r_count, 0);
	END_IF;

	(*UDP: IPC returns -1 if no data available or error occured,841 returns -1 if error occured and 0 if no data available*)
	CASE bytes_received OF
	-2147483648..-1: ; (* No data available or error occured *)
	 0: IF NOT udp_mode THEN (* TCP-Mode: socket wurde von remote geschlossen *)
			c_status := 253;
			c_ready := FALSE;
		END_IF;
	ELSE (* daten wurden empfangen *)
  		r_time := tx; (* Receive Timer ruecksetzen *)
		R_BUF.SIZE := INT_TO_UINT(r_offset + DINT_TO_UINT(bytes_received)); (* aktuelle buffersize eintragen *)
		IP_C.MAILBOX[1] := IP_C.MAILBOX[1] + 1; (* Receive Info *)
		IF IP_C.MAILBOX[1] = 0 THEN IP_C.MAILBOX[1] := 1; END_IF;

		(* ---------------------- Debug-Message ----------------------------*)
		(*IF _debug_enable THEN
			LOG_CL.NEW_MSG := 'IP_REC DATA: POS: ~1 : SIZE: ~2 TOTAL ~3 -IP_ID ~6';
			LOG_CL.PRINTF[1] := INT_TO_STRING(r_offset);
			LOG_CL.PRINTF[2] := INT_TO_STRING(r_count);
			LOG_CL.PRINTF[3] := UINT_TO_STRING(R_BUF.SIZE);
			LOG_CL.PRINTF[6] := INT_TO_STRING(debug_ID);
			LOG_MSG();
		END_IF;*)
		(* -----------------------------------------------------------------------------*)

	END_CASE
END_IF;

(* ---------------------------------------------- *)

IF S_BUF.SIZE > 0 THEN
	IF c_ready AND c_enable THEN
		IF NOT s_active AND IP_C.MAILBOX[2] = 0 THEN
			(* Gesamtanzahl an Bytes limitieren und uebergeben *)
			s_total := LIMIT(0,UINT_TO_INT(S_BUF.SIZE),r_max_size);
			s_cur_pos  := 0;
			s_cur_size := 0;
			s_start := TRUE; (* Daten kopieren und senden anstossen *)
			s_active := TRUE; (* Sende-Betrieb aktivieren *)
			(* ---------------------- Debug-Message ----------------------------*)
			(*IF _debug_enable THEN
				LOG_CL.NEW_MSG := 'IP_SEN INIT: TOTAL: ~1 -IP_ID ~6';
				LOG_CL.PRINTF[1] := INT_TO_STRING(S_TOTAL);
				LOG_CL.PRINTF[6] := INT_TO_STRING(debug_ID);
				LOG_MSG();
			END_IF;*)
			(* -----------------------------------------------------------------------------*)
		END_IF;

		IF s_done OR s_start THEN (* Daten senden aktiv *)

			s_start := FALSE;
			s_cur_pos := s_cur_pos + s_cur_size; (* neue Sende-Datenposition bestimmen *)
			IF s_total > s_cur_pos THEN (* weitere Daten zum senden vorhanden ? *)
				s_cur_size := s_total - s_cur_pos;
				s_cur_size := LIMIT(0, s_cur_size, s_max_size); (* Telegrammlänge begrenzen *)
				(* ---------------------- Debug-Message ----------------------------*)
				(*IF _debug_enable THEN
					LOG_CL.NEW_MSG := 'IP_SEN DATA: POS: ~1 : SIZE: ~2 TOTAL ~3 -IP_ID ~6';
					LOG_CL.PRINTF[1] := INT_TO_STRING(S_CUR_POS);
					LOG_CL.PRINTF[2] := INT_TO_STRING(S_CUR_SIZE);
					LOG_CL.PRINTF[3] := INT_TO_STRING(S_TOTAL);
					LOG_CL.PRINTF[6] := INT_TO_STRING(debug_ID);
					LOG_MSG();
				END_IF;*)
				(* -----------------------------------------------------------------------------*)
				s_time := tx; (* Send Timer ruecksetzen *)
				r_time := tx; (* Receive Timer ruecksetzen *)
				s_req := TRUE;

			ELSE
				(* keine weitere Sendedaten vorhanden -> Senden beenden *)
				s_req := FALSE;
				s_active := FALSE;
				S_BUF.SIZE := 0;
				(* ---------------------- Debug-Message ----------------------------*)
				(*IF _debug_enable THEN
					LOG_CL.NEW_MSG := 'IP_SEN FINISH -IP_ID ~6';
					LOG_CL.PRINTF[6] := INT_TO_STRING(debug_ID);
					LOG_MSG();
				END_IF;*)
				(* -----------------------------------------------------------------------------*)
			END_IF;
		END_IF;
	END_IF;
END_IF;

IF s_req THEN
	s_done := FALSE;
	IF udp_mode THEN
		bytes_sent := SysSockSendTo(socket, ADR(S_BUF.BUFFER[s_cur_pos]), s_cur_size, 0, ADR(sockaddr), SIZEOF(sockaddr));
	ELSE
		bytes_sent := SysSockSend(socket, ADR(S_BUF.BUFFER[s_cur_pos]), s_cur_size, 0);
	END_IF;

	CASE bytes_sent OF
	-2147483648..-1:	; (* ERROR: Noch nicht bereit um Daten aufzunehmen -> nächsten Zyklus wieder probieren *)
	 0: IF NOT udp_mode THEN (* TCP-Mode: socket wurde von remote geschlossen *)
			c_status := 253;
			c_ready := FALSE;
		END_IF;
	ELSE
		s_done := TRUE;
		s_cur_size := DINT_TO_INT(bytes_sent); (* Anzahl der wirklich versendeten Bytes übernehmen *)
		(* ---------------------- Debug-Message ----------------------------*)
		(*IF _debug_enable THEN
			LOG_CL.NEW_MSG := 'IP_SEN SEND_COUNT ~1 -IP_ID ~6';
			LOG_CL.PRINTF[1] := DINT_TO_STRING(s_cur_size);
			LOG_CL.PRINTF[6] := INT_TO_STRING(debug_ID);
			LOG_MSG();
		END_IF;*)
		(* -----------------------------------------------------------------------------*)
	END_CASE
END_IF;

(* ---------------------------------------------- *)

IF IP_C.R_OBSERVE = FALSE OR s_active THEN
    r_time := tx;
END_IF;

IF c_status = 0 AND tx - c_time > error_time AND c_enable AND NOT c_ready AND c_mode < 2 THEN (* Connect Timeout *)
	c_status := 255; (* Timeout-Fehler ausgeben *)
END_IF;
IF s_status = 0 AND tx - s_time > error_time AND s_active THEN (* Send Timeout *)
	s_status := 255; (* Timeout-Fehler ausgeben *)
END_IF;
IF r_status = 0 AND tx - r_time > error_time AND c_ready AND IP_C.R_OBSERVE THEN (* Receive Timeout *)
	r_status := 255; (* Timeout-Fehler ausgeben *)
END_IF;

IP_C.ERROR := OSCAT_BASIC.DWORD_OF_BYTE(c_status,s_status,r_status,0);

(* ---------------------- Debug-Message ----------------------------*)
(*IF  _debug_enable THEN
	IF (IP_C.ERROR <> debug_lasterror) THEN
		LOG_CL.NEW_MSG := 'IP_ERROR ~1 -IP_ID ~6';
		LOG_CL.PRINTF[1] := DWORD_TO_STRING(IP_C.ERROR);
		LOG_CL.PRINTF[6] := INT_TO_STRING(debug_ID);
		LOG_MSG();

		debug_lasterror := IP_C.ERROR;
		debug_last_id := debug_ID;
	END_IF;
END_IF;*)
(* -----------------------------------------------------------------------------*)

(* revision history
ks	18. oct. 2008	rev 1.0
	original version
ks	05. jan. 2009	rev 1.1
	zusätzlichen Parameter "Port" hinzugefügt, und Code bei Verbindungsaufbau angepasst
ks	28. feb. 2009	rev 1.2
	connect code angepasst und verkürzung der zyklen bei Send
ks	20. oct. 2009	rev 1.3
	network_buffer basis 0
ks	06. dec. 2009	rev 1.4
	receive_count MAILBOX[1]
ks	10. nov. 2010	rev 1.5
	send_pause MAILBOX[2] and receive_pause MAILBOX[3] 
ks	07. feb. 2011	rev 1.6
	Fehlercode 253 bei Remote-Verbindungsabbruch
ks	30. may. 2011	rev 1.7
	Fehler bei Empfangsüberwachung
ks	26. july. 2011	rev 1.8
	Error-Reset, diverse optimierungen 
ks	26. feb. 2012	rev 1.9
	Code-Optimierung für höhere kompatibilität

*)

END_FUNCTION_BLOCK

// POUs/CONVERT/IP4_TO_STRING
FUNCTION IP4_TO_STRING : STRING(15)
VAR_INPUT
	IP4 : DWORD;
END_VAR
VAR
	tmp : STRING(3);
END_VAR

(*
version 1.1	10. mar. 2009
programmer 	kurt
tested by	hugo

IP4_TO_STRING erzeugt eine IP Adresse als String aus einem DWORD..

*)

(* mask bits AND INSERT AT given position *)
tmp := BYTE_TO_STRING(DWORD_TO_BYTE(IP4));
IP4_TO_STRING := CONCAT('...', tmp);
tmp := BYTE_TO_STRING(DWORD_TO_BYTE(SHR(IP4,8)));
IP4_TO_STRING := INSERT(IP4_TO_STRING, tmp, 2);
tmp := BYTE_TO_STRING(DWORD_TO_BYTE(SHR(IP4,16)));
IP4_TO_STRING := INSERT(IP4_TO_STRING, tmp, 1);
tmp := BYTE_TO_STRING(DWORD_TO_BYTE(SHR(IP4,24)));
IP4_TO_STRING := CONCAT(tmp, IP4_TO_STRING);



(* revision history
hm	22. apr 2008	rev 1.0
	original version

hm	10. mar. 2009	rev 1.1
	improved code
*)

END_FUNCTION

// POUs/OTHER/IP_FIFO
FUNCTION_BLOCK IP_FIFO
VAR_IN_OUT
	FIFO : IP_FIFO_DATA;
	ID : BYTE;
	STATE : BYTE;
END_VAR
VAR
	tmp : INT;

	(*LOG_MSG : LOG_MSG;
	_debug_enable : BOOL := TRUE;*)

END_VAR

(*	version 1.0	18. oct. 2008
	programmer 	ks
	tested BY		ks

	IP_FIFO ist ein Zusatzbaustein füR die Zugriffsverwaltung auf IP_CONTROL
*)

IF NOT FIFO.INIT THEN
	FIFO.INIT := TRUE;
	FIFO.NW := 1;
	FIFO.NR := 1;
	FIFO.EMPTY := TRUE;
	FIFO.FULL := FALSE;
	FIFO.TOP := 128; (* Arraygroesse 1 bis x *)
	FIFO.MAX_ID := BYTE#1; (* maximale anzahl von Anmeldungen einer ID *)
END_IF;

(* wenn keine ID vorhanden dann die naechste freie ID zuteilen *)
IF ID = BYTE#00 THEN
	IF FIFO.ID < INT_TO_BYTE(FIFO.TOP) THEN
		ID := USINT_TO_BYTE(BYTE_TO_USINT(FIFO.ID) + USINT#1); (* ID +1 *)
		FIFO.ID := ID; (* ID eintragen *)
	    	(*####################  DEBUG-MESSAGE  ###################################*)
	    	(*IF _debug_enable THEN
	      		LOG_CL.NEW_MSG := 'FIFO: NEW ID:~1';
	      		LOG_CL.PRINTF[1]  := BYTE_TO_STRING(ID);
	      		LOG_MSG();
	    	END_IF;*)
	    	(*########################################################################*)
	ELSIF STATE < BYTE#200 THEN
		(*####################  DEBUG-MESSAGE  ###################################*)
		(*IF _debug_enable THEN
			LOG_CL.NEW_MSG := 'FIFO: OVERFLOW ADD ID';
			LOG_MSG();
		END_IF;*)
		(*########################################################################*)

		(* sollte nie passieren ! -> es sind zuviele teilnehmer angemeldet *)
		(* es wird keine Nummer vergeben und alle anfragen werden negativ beantwortet *)
		STATE := BYTE#255;
		RETURN;
	END_IF;
END_IF;

IF STATE = BYTE#1 AND NOT FIFO.FULL THEN (* Anmelden *)
	(* nur eintragen wenn maximale anzahl nicht ueberschritten wurde *)
	tmp := BYTE_TO_INT(ID);
	IF FIFO.Y[tmp] < FIFO.MAX_ID THEN
		FIFO.Y[tmp] := USINT_TO_BYTE(BYTE_TO_USINT(FIFO.Y[tmp]) + USINT#1); (* IP_ID Zähler +1 *)
		tmp := FIFO.NW; (* geht bei mir leider nicht anders *)
		FIFO.X[tmp] := ID;
		IF FIFO.NW = FIFO.TOP THEN FIFO.NW := 1; ELSE FIFO.NW := FIFO.NW + 1; END_IF;
		FIFO.FULL := FIFO.NW = FIFO.NR;
		FIFO.EMPTY := FALSE;
		STATE := BYTE#2; (* weiterschalten auf "Warten auf Freigabe" *)
		(*####################  DEBUG-MESSAGE  ###################################*)
		(*IF _debug_enable THEN
			LOG_CL.NEW_MSG := 'FIFO: ADD ID:~1';
			LOG_CL.PRINTF[1]  := BYTE_TO_STRING(ID);
			LOG_MSG();
		END_IF;*)
		(*########################################################################*)

	END_IF;
END_IF;

IF STATE = BYTE#2 AND NOT FIFO.EMPTY THEN (* check current stack element *)
	tmp := FIFO.NR; (* geht bei mir leider nicht anders *)
	IF ID = FIFO.X[tmp] THEN
	STATE := BYTE#3; (* weiterschalten auf "Zugriffsfreigabe" *)
	END_IF;
END_IF;

IF STATE = BYTE#4 AND NOT FIFO.EMPTY THEN (* remove from stack *)
	tmp := FIFO.NR; (* geht bei mir leider nicht anders *)
	IF ID = FIFO.X[tmp] THEN
		tmp := BYTE_TO_INT(ID); (* geht bei mir leider nicht anders *)
		FIFO.Y[tmp] := USINT_TO_BYTE(BYTE_TO_USINT(FIFO.Y[tmp]) - USINT#1); (* ID Zähler -1 *)
		IF FIFO.NR = FIFO.TOP THEN FIFO.NR := 1; ELSE FIFO.NR := FIFO.NR + 1; END_IF;
		FIFO.EMPTY := FIFO.NR = FIFO.NW;
		FIFO.FULL := FALSE;
		(*####################  DEBUG-MESSAGE  ###################################*)
		(*IF _debug_enable THEN
			LOG_CL.NEW_MSG := 'FIFO: REMOVE ID:~1';
			LOG_CL.PRINTF[1]  := BYTE_TO_STRING(ID);
			LOG_MSG();
		END_IF;*)
		(*########################################################################*)
	END_IF;
	STATE := BYTE#5; (* "Remove done" *)
END_IF;

(* revision history
ks	18. oct. 2008	rev 1.0
	original version

*)

END_FUNCTION_BLOCK

// POUs/DEMO/DLOG_FILE_CSV_SMTP_DEMO
PROGRAM DLOG_FILE_CSV_SMTP_DEMO
VAR
	cur_dt: DT;
	enable: BOOL := TRUE;
	trig_t : TIME := T#5s;
	trig_m : BOOL;
	error_c: DWORD;
	error_t: BYTE;
	auto_close: TIME := T#10s;

	x1: DLOG_DT;
	x2 : DLOG_REAL;
	x3 : DLOG_DINT;
	x4 : DLOG_BOOL;
	x5: DLOG_STRING;
	x : DLOG_DATA;
	RTC_2: oscat_basic.RTC_2;
	DLOG_STORE_FILE_CSV : DLOG_STORE_FILE_CSV;
	GEN_SIN_1: oscat_basic.GEN_SIN;
	COUNT_DR: oscat_basic.COUNT_DR;

	DLOG_FILE_TO_SMTP: DLOG_FILE_TO_SMTP;
	smtp_timeout: TIME := T#30s;
	smtp_error_t: BYTE;
	smtp_error_c: DWORD;
	smtp_busy: BOOL;
	smtp_done: BOOL;
	smtp_dti: DT;
	smtp_dti_offset: INT := 60;
	smtp_server: STRING := '110876022:oscat123456@mail.gmx.net';
	smtp_mailfrom: STRING := 'oscat@gmx.net;Station_01';
	smtp_mailto: STRING(OSCAT_BASIC.STRING_LENGTH) := 'oscat@gmx.net';
	smtp_subject: STRING := 'Das ist der Betreff';
	smtp_body: STRING(OSCAT_BASIC.STRING_LENGTH) := 'Das ist der Email-Text';
	smtp_delete: BOOL := TRUE;
	smtp_retry: INT := 0;
	smtp_retry_time: TIME := T#60s;
END_VAR

VAR RETAIN
	save_data : DLOG_SAVE;
END_VAR
VAR // added by the converter: edge detectors and wires of the graphical bodies
    _w1, _w2 : ANY;
END_VAR

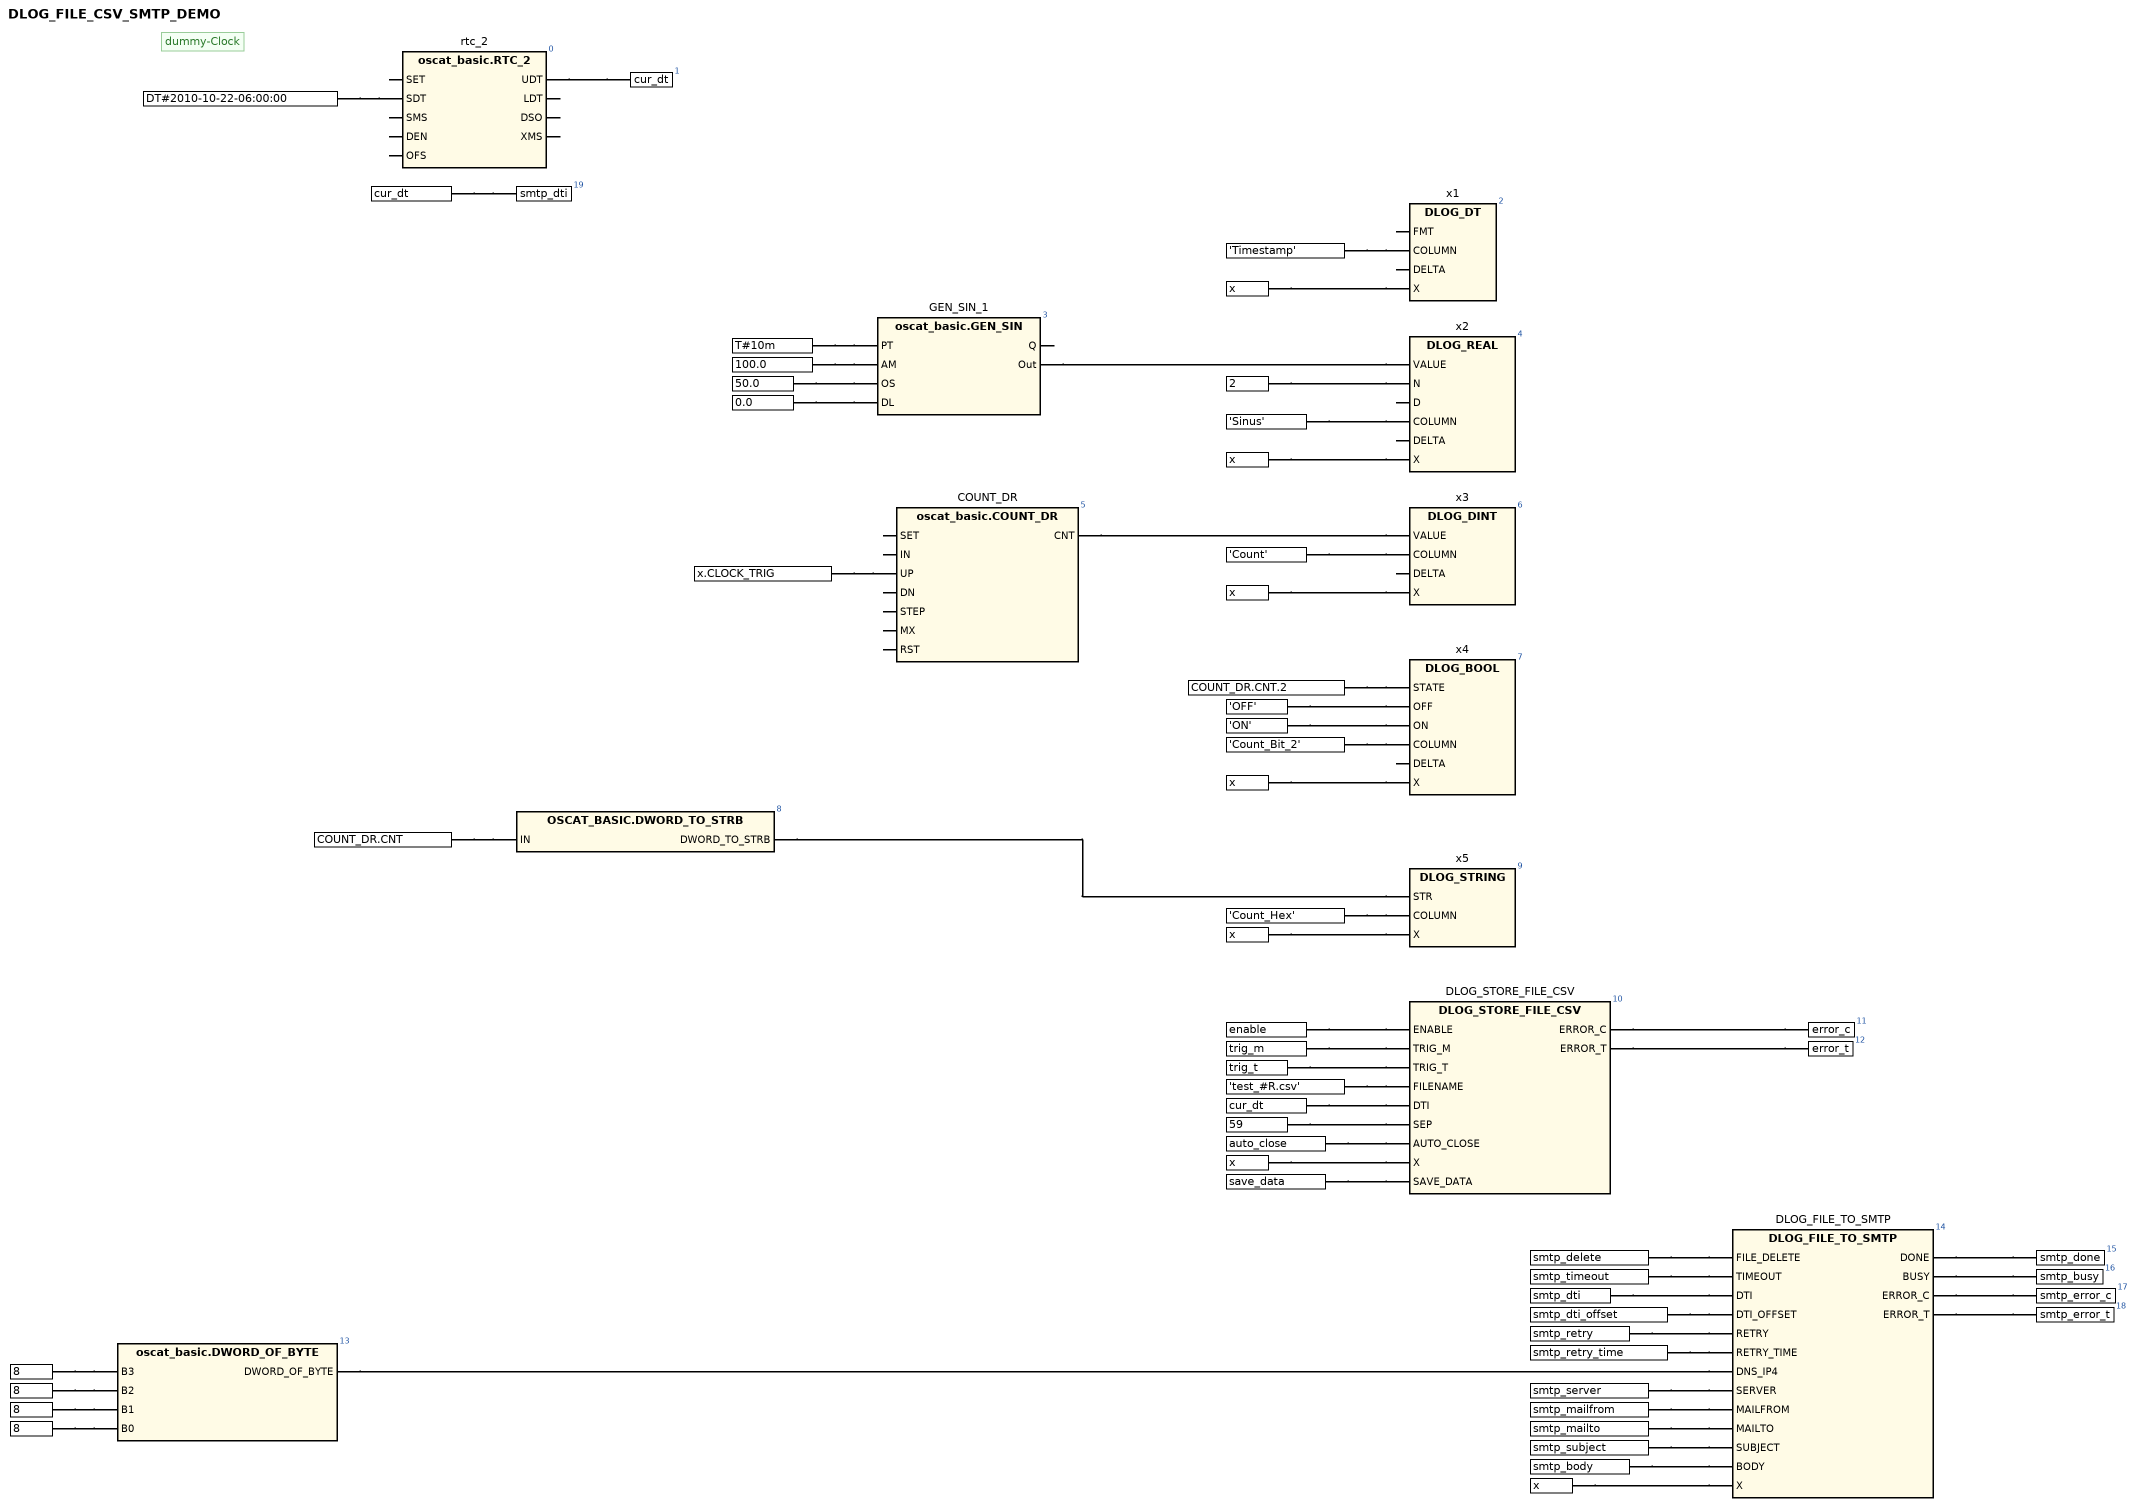
// dummy-Clock
rtc_2(SDT := DT#2010-10-22-06:00:00); // oscat_basic.RTC_2
cur_dt := rtc_2.UDT;
x1(COLUMN := 'Timestamp', X := x); // DLOG_DT
GEN_SIN_1(PT := T#10m, AM := 100.0, OS := 50.0, DL := 0.0); // oscat_basic.GEN_SIN
x2(VALUE := GEN_SIN_1.Out, N := 2, COLUMN := 'Sinus', X := x); // DLOG_REAL
COUNT_DR(UP := x.CLOCK_TRIG); // oscat_basic.COUNT_DR
x3(VALUE := COUNT_DR.CNT, COLUMN := 'Count', X := x); // DLOG_DINT
x4(STATE := COUNT_DR.CNT.2, OFF := 'OFF', ON := 'ON', COLUMN := 'Count_Bit_2', X := x); // DLOG_BOOL
_w1 := OSCAT_BASIC.DWORD_TO_STRB(IN := COUNT_DR.CNT);
x5(STR := _w1, COLUMN := 'Count_Hex', X := x); // DLOG_STRING
DLOG_STORE_FILE_CSV(
    ENABLE := enable,
    TRIG_M := trig_m,
    TRIG_T := trig_t,
    FILENAME := 'test_#R.csv',
    DTI := cur_dt,
    SEP := 59,
    AUTO_CLOSE := auto_close,
    X := x,
    SAVE_DATA := save_data);
error_c := DLOG_STORE_FILE_CSV.ERROR_C;
error_t := DLOG_STORE_FILE_CSV.ERROR_T;
_w2 := oscat_basic.DWORD_OF_BYTE(B3 := 8, B2 := 8, B1 := 8, B0 := 8);
DLOG_FILE_TO_SMTP(
    FILE_DELETE := smtp_delete,
    TIMEOUT := smtp_timeout,
    DTI := smtp_dti,
    DTI_OFFSET := smtp_dti_offset,
    RETRY := smtp_retry,
    RETRY_TIME := smtp_retry_time,
    DNS_IP4 := _w2,
    SERVER := smtp_server,
    MAILFROM := smtp_mailfrom,
    MAILTO := smtp_mailto,
    SUBJECT := smtp_subject,
    BODY := smtp_body,
    X := x);
smtp_done := DLOG_FILE_TO_SMTP.DONE;
smtp_busy := DLOG_FILE_TO_SMTP.BUSY;
smtp_error_c := DLOG_FILE_TO_SMTP.ERROR_C;
smtp_error_t := DLOG_FILE_TO_SMTP.ERROR_T;
smtp_dti := cur_dt;

END_PROGRAM

// POUs/DATA_LOG/DLOG_FILE_TO_SMTP
FUNCTION_BLOCK DLOG_FILE_TO_SMTP
VAR_IN_OUT
	SERVER : STRING;
	MAILFROM : STRING;
	MAILTO : STRING(OSCAT_BASIC.STRING_LENGTH);
	SUBJECT : STRING;
	BODY : STRING(OSCAT_BASIC.STRING_LENGTH);
	X : DLOG_DATA;
END_VAR
VAR_INPUT
	FILE_DELETE : BOOL;
	TIMEOUT : TIME := T#30s;
	DTI : DT;
	DTI_OFFSET : INT;
	RETRY : INT;
	RETRY_TIME : TIME := T#30s;
	DNS_IP4 : DWORD;
END_VAR
VAR_OUTPUT
	DONE : BOOL;
	BUSY : BOOL;
	ERROR_C : DWORD;
	ERROR_T : BYTE;
END_VAR
VAR
	UCBD : UNI_CIRCULAR_BUFFER_DATA;
	UCB : UNI_CIRCULAR_BUFFER;
	SMTP_CLIENT : SMTP_CLIENT;
	WT_1 : TON;
	ftrig_old : BOOL;
	files : STRING(OSCAT_BASIC.STRING_LENGTH);
	step : INT;
	smtp_busy : BOOL;
	smtp_done : BOOL;
	cnt : INT;

	(*LOG_MSG : LOG_MSG;
	_debug_enable : BOOL := TRUE;*)
END_VAR

(*
version 1.3		21. mar. 2016
programmer		ks
tested by			ks

DLOG_FILE_TO_SMTP der Baustein versendet die vom DLOG_STORE_FILE_CSV erzeugten Dateien als Email
*)

(* neue Filenamen speichern *)
IF X.NEW_FILE_RTRIG AND ftrig_old = FALSE THEN
	UCBD.D_HEAD := 1;
	UCBD.D_MODE := 1;
	UCBD.D_STRING := X.NEW_FILE;
	UCB(DATA:=UCBD); (* Daten eintragen *)
END_IF;
ftrig_old := X.NEW_FILE_RTRIG;

CASE step OF

00:	IF UCBD.BUF_COUNT > 0 AND smtp_busy = FALSE THEN
		UCBD.D_MODE := 12; (* Daten lesen und löschen *)
		UCB(DATA:=UCBD);
		files := UCBD.D_STRING;
		IF FILE_DELETE THEN
			files := CONCAT(files,';#DEL#');
		END_IF;
		cnt := RETRY;
		step := 10;

		(*####################  DEBUG-MESSAGE  ###################################*)
		(*IF _debug_enable THEN
			LOG_CL.NEW_MSG := 'F_T_SMTP: Auftrag aktiv /file: ~2';
			LOG_CL.PRINTF[2] := files;
			LOG_MSG();
		END_IF;*)
		(*########################################################################*)

	END_IF;

10:	IF smtp_busy = FALSE THEN
		IF smtp_done THEN
			(*####################  DEBUG-MESSAGE  ###################################*)
			(*IF _debug_enable THEN
				LOG_CL.NEW_MSG := 'F_T_SMTP: Auftrag OK /file: ~2';
				LOG_CL.PRINTF[2] := files;
				LOG_MSG();
			END_IF;*)
			(*########################################################################*)
			step := 0;
		ELSE
			step := 20; (* pause nach error *)
		END_IF;
	END_IF;

20:	IF WT_1.Q THEN (* Wartezeit *)
		cnt := cnt - 1;
		IF RETRY = 0 THEN (* Transfer unbegrenzt wiederholen *)
			(*####################  DEBUG-MESSAGE  ###################################*)
			(*IF _debug_enable THEN
				LOG_CL.NEW_MSG := 'F_T_SMTP: Auftrag unbegrenzt wiederholen /file: ~2';
				LOG_CL.PRINTF[2] := files;
				LOG_MSG();
			END_IF;*)
			(*########################################################################*)
			step := 10; (* Transfer wiederholen *)
		ELSIF cnt >= 0 THEN
			(*####################  DEBUG-MESSAGE  ###################################*)
			(*IF _debug_enable THEN
				LOG_CL.NEW_MSG := 'F_T_SMTP: Auftrag wiederholen /cnt: ~1 /file: ~2';
				LOG_CL.PRINTF[1] := INT_TO_STRING(cnt);
				LOG_CL.PRINTF[2] := files;
				LOG_MSG();
			END_IF;*)
			(*########################################################################*)
			step := 10; (* Transfer wiederholen *)
		ELSE
			(*####################  DEBUG-MESSAGE  ###################################*)
			(*IF _debug_enable THEN
				LOG_CL.NEW_MSG := 'F_T_SMTP: Auftrag verworfen /file: ~2';
				LOG_CL.PRINTF[2] := files;
				LOG_MSG();
			END_IF;*)
			(*########################################################################*)
			step := 0; (* Auftrag verwerfen *)
		END_IF;
	END_IF;

END_CASE;

BUSY := step = 10;
DONE := step = 0;
WT_1(IN:= step = 20, PT:= RETRY_TIME);

SMTP_CLIENT(
	ACTIVATE:= BUSY,
	TIMEOUT:= TIMEOUT,
	DTI:= DTI,
	DTI_OFFSET:= DTI_OFFSET,
	DNS_IP4:= DNS_IP4,
	SERVER:= SERVER,
	MAILFROM:= MAILFROM,
	MAILTO:= MAILTO,
	SUBJECT:= SUBJECT,
	BODY:= BODY,
	FILES:= FILES,
	DONE=> smtp_done,
	BUSY=> smtp_busy
	);

(* Fehlerauswertung *)
IF SMTP_CLIENT.ERROR_T <> BYTE#0 THEN
	ERROR_C := SMTP_CLIENT.ERROR_C;
	ERROR_T := SMTP_CLIENT.ERROR_T;
ELSIF UCBD.BUF_DATA_LOST > UDINT#0 THEN
	ERROR_C := DWORD#2; (* Fehler: Bufferüberlauf - Datenmenge reduzieren *)
	ERROR_T := BYTE#6; 	(* Type: Buffer *)
ELSIF UCBD.BUF_USED_MAX > USINT#90 THEN
	ERROR_C := DWORD#1; (* Warnung: Buffer auslastung > 90% *)
	ERROR_T := BYTE#6;	(* Type: Buffer *)
ELSE
	ERROR_C := DWORD#0;
	ERROR_T := BYTE#0;
END_IF;

(* revision history

ks	01. jan. 2011	rev 1.0
	original version

ks	28. apr. 2011	rev 1.1
	stringfehler bei option 'file_delete'

ks	26. jul. 2011	rev 1.2
    codeoptimierung D_MODE 12

ks	21. mar. 2016	rev 1.3
	fehlermeldungen hinzugefügt
	fehler in RETRY korrigiert

*)

END_FUNCTION_BLOCK

// POUs/NETWORK/SMTP_CLIENT
FUNCTION_BLOCK SMTP_CLIENT
VAR_INPUT
	ACTIVATE : BOOL;
	TIMEOUT : TIME;
	DTI : DT;
	DTI_OFFSET : INT;
	DNS_IP4 : DWORD;
END_VAR
VAR_OUTPUT
	DONE : BOOL;
	BUSY : BOOL;
	ERROR_C : DWORD;
	ERROR_T : BYTE;
END_VAR
VAR_IN_OUT
	SERVER : STRING;
	MAILFROM : STRING;
	MAILTO : STRING(OSCAT_BASIC.STRING_LENGTH);
	SUBJECT : STRING;
	BODY : STRING(OSCAT_BASIC.STRING_LENGTH);
	FILES : STRING(OSCAT_BASIC.STRING_LENGTH);
END_VAR
VAR
	IP_C : IP_C; (* IP_Control Verwaltungsstruktur *)
	S_BUF : NETWORK_BUFFER;
	R_BUF : NETWORK_BUFFER;
	F_BUF : NETWORK_BUFFER;
	URL_DATA : url;
	DNS_CLIENT : DNS_CLIENT;
	IPC : IP_CONTROL;
	FS : FILE_SERVER;
	FSD : FILE_SERVER_DATA;
	BASE64_ENCODE_STR : BASE64_ENCODE_STR;
	BASE64_ENCODE_STREAM : BASE64_ENCODE_STREAM;
	fpd : FILE_PATH_DATA;
	MD5_CRAM_AUTH : MD5_CRAM_AUTH;
	MD5_RUN : BOOL;
	activate_last : BOOL;
	step : INT;
	snd_step : INT;
	str1 : STRING(OSCAT_BASIC.STRING_LENGTH);
	str2 : STRING(OSCAT_BASIC.STRING_LENGTH);
	str3 : STRING;
	snd_text :	STRING(OSCAT_BASIC.STRING_LENGTH);
	snd_lf_cnt : INT;
	rcv_text :	STRING(OSCAT_BASIC.STRING_LENGTH);
	rcv_s : STRING(3);
	rcv_state : INT;
	auth_names : STRING := ' PLAIN; LOGIN; CRAM-MD5';
	auth_names_tls : STRING := ' PLAIN; LOGIN; CRAM-MD5;STARTTLS';
	auth_state : BYTE;
	TON_WAIT : TON;
	last_step : INT;
	next_step : INT;
	timeout2 : TIME;
	timeout3 : TIME;
	last_block : BOOL;
	file_delete : BOOL;
	esmtp : BOOL;
	cnt1 : INT;
	cnt2 : INT;
	cnt3 : INT;
	cnt4 : INT;
	idx1 : INT;
	idx2 : INT;
	idx3 : INT;
	snd_idx : INT;
	snd_enable : BOOL;
	i1 : INT;
	b64_done : BOOL;
	b64_start : BOOL;
	b64_max : UINT := 2880; (* short = 960 / long = 2880 *)
	b64_buf1 : ARRAY [0..47] OF BYTE;
	b64_buf2 : ARRAY [0..63] OF BYTE;
	b64_size1 : INT;
	b64_size2 : INT;
	b64_lf : BOOL;
	b64_str1	: STRING(144);
	b64_str2	: STRING(192);
	md5_user : STRING(64);
	md5_password : STRING(64);
	md5_b64_ts : STRING(64);
	md5_auth_key : STRING(192);
	ip_c_red_disable : BOOL; (* IP_CONTROL - Remote Disconnect Error unterdrücken *)
	ssl_mode :	BYTE;(*SSL/TLS Mode -   0 = off / 1 = SSL / 2 = TLS*)

	(*LOG_MSG : LOG_MSG;
	_debug_enable : BOOL := TRUE;*)
END_VAR

(*
version 1.7		18. aug 2016
programmer		ks
tested by		ks

SMTP_CLIENT versendet Email an verschiedene Emailadressen mit optionalen Dateianhängen.



mögliche Rückgabecodes:

Grad der Schwere
 
Die erste Stelle des Rückgabecodes gibt den Grad der Schwere an:
1yz Vorläufige positive Antwort
2yz Antwort über positiven Abschluss 
3yz Positive Zwischenantwort 
4yz Antwort über vorübergehenden negativen Abschluss 
5yz Permanente negative Antwort 
 
Die zweite Stelle gibt die Kategorie der Antwort an: 
x0z Syntaxfehler 
x1z Information 
x2z Verbindung 
x3z Nicht festgelegt 
x4z Nicht festgelegt 
x5z Mail-System 
 
Die dritte Stelle dient zur genaueren Bestimmung der Kategorie. 

Betriebsprotokolle enthalten folgende Codes: 
211 	Systemstatus oder Hilfe-Antwort des Systems  
214 	Hilfe-Nachricht - Informationen zur Verwendung des Empfängers oder zur  
      	Bedeutung eines bestimmten nicht standardmäßigen Befehls; wobei  
      	diese Antwort nur für Personen hilfreich ist, nicht für Systeme 
220 	Service ready (Dienst bereit) 
221 	Service closing transmission channel (Dienst schließt Übertragungskanal) 
235  Authentication succeeded (Authentifizierung erfolgreich)
250 	Requested mail action okay, completed (angeforderte Mail-Maßnahme ok und abgeschlossen) 
251 	User not local; will forward to (Benutzer nicht lokal; Weiterleitung an) 
252 	Cannot VRFY user, but will accept message and attempt delivery (kann Benutzer nicht überprüfen, aber akzeptiert Nachricht und versucht Auslieferung) 
354 	Start mail input; end with. (Mail-Eingabe starten; Ende mit .) 
421 	Service not available, closing transmission channel 	(Dienst nicht verfügbar, Übertragungskanal wird geschlossen) diese Antwort kann auf jeden Befehl folgen, wenn der Dienst weiß, dass er beendet werden muss 
450 	Requested mail action not taken: mailbox unavailable (angeforderte E-Mail-Maßnahme nicht ausgeführt, Mailbox nicht  verfügbar) - z. B. weil Mailbox besetzt 
451	 Requested action aborted: local error in processing (angeforderte Maßnahme abgebrochen: lokaler Fehler bei der Verarbeitung) 
452 	Requested action not taken: insufficient system storage (angeforderte Maßnahme abgebrochen: Systemspeicher nicht ausreichend) 
500 	Syntax error, command unrecognized (Syntaxfehler, Befehl nicht erkannt) - z. B. weil Befehlszeile zu lang 
501 	Syntax error in parameters or arguments (Syntaxfehler in Parametern oder Argumenten) 
502 	Command not implemented (Befehl nicht implementiert) 
504 	Command parameter not implemented (Befehlsparameter nicht implementiert) 
550 	Requested action not taken: mailbox unavailable (Angeforderte Maßnahme nicht ausgeführt: Mailbox nicht verfügbar) 
551 	User not local; please try (Benutzer nicht lokal; versuchen Sie es mit) 
552 	Requested mail action aborted: exceeded storage allocation (angeforderte Mail-Maßnahme abgebrochen: Speicherplatzzuweisung überschritten) 
553 	Requested action not taken: mailbox name not allowed (angeforderte Maßnahme nicht ausgeführt: Mailboxname nicht zulässig) 
554 	Transaction failed (Transaktion fehlgeschlagen) 

534		Google Sonderbehandlung
		https://www.google.com/settings/security/lesssecureapps and set "Access for less secure apps" to ON

#########################
ERROR_T

1 = DNS_CLIENT
2 = SMTP Steuerkanal
4 = FILE_SERVER
5 = Ablaufstörung
#########################

*)

CASE step OF

00:
	IF ACTIVATE AND NOT activate_last THEN
		TIMEOUT := MAX(T#10s,TIMEOUT);
		timeout2 := TIMEOUT + T#1s;
		timeout3 := TIMEOUT / 2;
		DONE := FALSE;
		ip_c_red_disable := FALSE;
		ERROR_C := DWORD#0;
		ERROR_T := BYTE#0;
		FSD.ERROR := BYTE#0;
		file_delete := FALSE;
		URL_DATA := STRING_TO_URL(STR:=SERVER,DEFAULT_PROTOCOL:='',DEFAULT_PATH:='/');
		idx1 := FIND(URL_DATA.USER,'%'); (* % Zeichen auf @ ändern *)
		IF idx1 > 0 THEN
			URL_DATA.USER := REPLACE(URL_DATA.USER,'@',1,idx1);
		END_IF;
		esmtp := LEN(URL_DATA.PASSWORD) > 0; (* SMTP oder ExtendedSMTP *)
		step := 10;
	END_IF;

10:
	IF DNS_CLIENT.DONE THEN
		step := 20;
	ELSIF DNS_CLIENT.ERROR <> DWORD#0 THEN
		ERROR_C := DNS_CLIENT.ERROR;
		ERROR_T := BYTE#1;
		step := 980;
	END_IF;

20:	(* SMTP Kommunikation einrichten *)
	IF FIND(';SSL;ssl;Ssl', URL_DATA.PROTOCOL) > 1 THEN
		ssl_mode := BYTE#1;
		IP_C.C_PORT := SEL(URL_DATA.PORT = WORD#0,URL_DATA.PORT,WORD#465); (* Portnummer eintragen *)
		IP_C.MAILBOX[16] := BYTE#1; (* SSL Mode freigeben *)
	ELSIF FIND(';TLS;tls;Tls', URL_DATA.PROTOCOL) > 1 THEN
		ssl_mode := BYTE#2;
		IP_C.C_PORT := SEL(URL_DATA.PORT = WORD#0,URL_DATA.PORT,WORD#587); (* Portnummer eintragen *)
		IP_C.MAILBOX[16] := BYTE#0; (* noch kein SSL Mode*)
	ELSE
		ssl_mode := BYTE#0;
		IP_C.C_PORT := SEL(URL_DATA.PORT = WORD#0,URL_DATA.PORT,WORD#25); (* Portnummer eintragen *)
		IP_C.MAILBOX[16] := BYTE#0; (* kein SSL Mode*)
	END_IF;

  	IP_C.C_IP := DNS_CLIENT.IP4; (* IP eintragen *)
  	IP_C.C_MODE := BYTE#0; (* Mode: TCP+ACTIV+PORT *)
  	IP_C.TIME_RESET := TRUE; (* Zeitueberwachung rücksetzen *)
  	IP_C.C_ENABLE := TRUE; (* Verbindungsaufbau freigeben *)
  	IP_C.R_OBSERVE := TRUE; (* Empfangsueberwachung *)
	IP_C.MAILBOX[3] := BYTE#0; (* IP Empfang wieder freigeben *)
	R_BUF.SIZE := UINT#0;
	snd_enable := TRUE; (* sofortiges senden erlauben *)
	snd_idx := 0;
	step := 30;

30:	
	IF rcv_state = 220 THEN (* 220 = Service ready *)
		IF esmtp THEN
			snd_text := 'EHLO OSCAT'; (* ExtendedSMTP *)

			str1:= SEL(ssl_mode = BYTE#2,auth_names,auth_names_tls);
			auth_state := BYTE#0;
			idx2 := 1900;

			next_step := 40;
		ELSE
			snd_text := 'HELO OSCAT'; (* SMTP *)
			next_step := 90;
		END_IF;
		snd_lf_cnt := 1;
	END_IF;

40:	
	IF rcv_state = 250 THEN
		(* 250 = Requested mail action okay, complete
			1. bei manchen Providern wird bei SSL kein AUTH verfahren ausgeben.
			2. Da die 250 xxx Meldungen vom manchen SMTP-Servern mit mehr als einem Telegramme versendet
		       werden muss alternativ über Zeitüberwachung eine SSL Sonderbehandlung durchgeführt werden *)
		IF ssl_mode >= BYTE#1 AND TON_WAIT.ET > T#1s THEN
			rcv_text := '250-AUTH LOGIN'; (* AUTH vortäuschen *)

        	(*####################  DEBUG-MESSAGE  ###################################*)
			(*IF _debug_enable THEN
				LOG_CL.NEW_MSG := 'SMTP: PROBLEM /rcv_text ~1';
				LOG_CL.PRINTF[1] := rcv_text;
				LOG_MSG();
			END_IF;*)
			(*########################################################################*)

		END_IF;

		IF FIND(rcv_text,'AUTH') > 0 THEN (* BUGFIX  !*)
			IP_C.MAILBOX[3] := BYTE#1; (* IP Empfang blockieren bis Daten überprüft wurden *)
			idx1 := 0;
			step := 50;
		END_IF;

	END_IF;

50:
	str2 := ELEMENT_GET(59, idx1, str1); (* Trennzeichen >;< *)

	(*####################  DEBUG-MESSAGE  ###################################*)
	(*IF _debug_enable THEN
		LOG_CL.NEW_MSG := 'ST s1>~1< s2>~2< i1>~2< ~3';
		LOG_CL.PRINTF[1] := str1;
		LOG_CL.PRINTF[2] := str2;
		LOG_CL.PRINTF[3] := INT_TO_STRING(idx1);
		LOG_CL.PRINTF[4] := rcv_text;
		LOG_MSG();
	END_IF;*)
	(*########################################################################*)

	IF LEN(str2) > 0 THEN
		IF FIND(rcv_text,str2) > 0 THEN
			auth_state := OSCAT_BASIC.BIT_LOAD_B(auth_state, TRUE, idx1);
			str3 := str2; (* aktuellen AUTH-Type Namen sichern *)
			idx2 := 1000 + (idx1 * 100); (* Schritt berechnen *)
		END_IF;
		idx1 := idx1 + 1;
	ELSE
		IF auth_state <> BYTE#0 THEN (* AUTH-Type gefunden *)
			IP_C.MAILBOX[3] := BYTE#0; (* IP Empfang wieder freigeben *)
			(* mit den jeweiligen Authentifizierung Schritten fortfahren:
			   1000 = PLAIN / 1100 = LOGIN / 1200 = CRAM-MD5 / 1300 TLS *)
			step := idx2;
		ELSE
			idx1 := 0;
			rcv_text := '';
			IP_C.MAILBOX[3] := BYTE#0; (* IP Empfang wieder freigeben *)
			step := 40; (* warten auf nächste 250 auth meldung *)
		END_IF;
	END_IF;

	(*####################  DEBUG-MESSAGE  ###################################*)
	(*IF _debug_enable THEN
		LOG_CL.NEW_MSG := 'SMTP: /auth ~1 /idx1 ~2 /idx2 ~3 /str3 ~4 /LEN ~5 /step ~6 /str1 ~7';
		LOG_CL.PRINTF[1] := BYTE_TO_STRING(auth_state);
		LOG_CL.PRINTF[2] := INT_TO_STRING(idx1);
		LOG_CL.PRINTF[3] := INT_TO_STRING(idx2);
		LOG_CL.PRINTF[4] := str3;
		LOG_CL.PRINTF[5] := INT_TO_STRING(LEN(str2));
		LOG_CL.PRINTF[6] := INT_TO_STRING(step);
		LOG_CL.PRINTF[7] := str1;
		LOG_MSG();
	END_IF;*)
	(*########################################################################*)

 (* ++++++++++++++++++++++++++++++++++++++++++++++++++++++*)

90:
	IF rcv_state = 235 OR rcv_state = 250 THEN (* 235 = Authentication successful / 250 Requested mail action okay *)
		str2 := MAILFROM;
		str1 := ELEMENT_GET(59, 0, str2);(* MAILFROM lesen , Trennzeichen >;< *)
		snd_text := INSERT('MAIL FROM: <>', str1, 12);
		str3 := REPLACE(snd_text, 'From', 9, 1); (* 'MAIL FROM' durch "From" ersetzen und zwischenspeichern *)
		next_step := 95;
		cnt1 := ELEMENT_COUNT(35, MAILTO); (* Trennzeichen >#< , Anzahl der Blöcke bestimmen *)
		cnt2 := 0;
	END_IF;

95:	
	IF rcv_state = 250 THEN (* 250 = Requested mail action okay *)
		IF cnt2 < cnt1 THEN
			str1 := ELEMENT_GET(35, cnt2, MAILTO);(* Trennzeichen >#< *)
			cnt3 := ELEMENT_COUNT(59, str1); (* Trennzeichen >;< , Anzahl der Sub-Blöcke bestimmen *)
			cnt4 := 0;
			cnt2 := cnt2 + 1;
			step := 100; (* Blockinhalt auswerten *)
		ELSE
			step := 110; (* alle Blöcke bearbeitet *)
		END_IF;
	END_IF;

100:
	IF rcv_state = 250 THEN (* 250 = Requested mail action okay *)
		IF cnt4 < cnt3 THEN
			str2 := ELEMENT_GET(59, cnt4, str1); (* Trennzeichen >;< *)
			snd_text := INSERT('RCPT TO: <>', str2, 10);
			cnt4 := cnt4 + 1;
			next_step := 100;
		ELSE
			step := 95;
		END_IF;
	END_IF;

110:
	IF rcv_state = 250 THEN (* 250 = Requested mail action okay *)
		snd_text := 'DATA';
		next_step := 120;
	END_IF;

120:
	IF rcv_state = 354 THEN (* 354 = Start mail input; end with. *)
		snd_enable := FALSE;
		str2 := MAILFROM;
		str1 := ELEMENT_GET(59, 1, str2);(* Angezeigter Name lesen , Trennzeichen >;< *)
		IF LEN(str1) > 0 THEN
			str2 := INSERT('"" ', str1, 1);
			snd_text := INSERT(str3, str2, 6);
		ELSE
			snd_text := str3;
		END_IF;
		cnt2 := 0;
		cnt1 := MIN(2,cnt1); (* BlindCopy Block ausblenden *)
		step := 200;
	END_IF;

200:
	IF snd_step = 0 THEN
		IF cnt2 < cnt1 THEN
			str1 := ELEMENT_GET(35, cnt2, MAILTO);(* Trennzeichen >#< *)
			cnt3 := ELEMENT_COUNT(59, str1); (* Trennzeichen >;< , Anzahl der Sub-Blöcke bestimmen *)
			cnt4 := 0;
			cnt2 := cnt2 + 1;
			str3 := SEL(cnt2 = 1,'Cc: <>','To: <>');
			step := 205; (* Blockinhalt auswerten *)
		ELSE
			step := 210; (* alle Blöcke bearbeitet *)
		END_IF;
	END_IF;

205:
	IF snd_step = 0 THEN
		IF cnt4 < cnt3 THEN
			str2 := ELEMENT_GET(59, cnt4, str1); (* Trennzeichen >;< *)
			snd_text := INSERT(str3, str2, 5);
			cnt4 := cnt4 + 1;
		ELSE
			step := 200;
		END_IF;
	END_IF;

210:
	IF snd_step = 0 THEN
		snd_text := CONCAT('Subject: ',SUBJECT);
		step := 220;
	END_IF;

220:
	IF snd_step = 0 THEN
		DTI := UDINT_TO_DT(DT_TO_UDINT(DTI) + INT_TO_UDINT(- DTI_OFFSET * 60)); (* Minuten-Offset auf Sekunden umrechnen und addieren *)
		IF esmtp THEN (* ESMTP Format >Date: Thu, 21 May 1998 05:33:29 -0700< *)
			str2 := ';Mon;Tue;Wed;Thu;Fri;Sat;Sun';
			str1 := ELEMENT_GET(59, OSCAT_BASIC.DAY_OF_WEEK(DT_TO_DATE(DTI)), str2);
			snd_text := CONCAT('Date: ',str1);
			str1 := OSCAT_BASIC.DT_TO_STRF(DTI, 0, ', #H #E #A #N:#R:#T +0000', 1);
			snd_text := CONCAT(snd_text,str1);
		ELSE (* SMTP Format >Date: 21 May 98 05:33:29< *)
			snd_text := OSCAT_BASIC.DT_TO_STRF(DTI, 0, 'Date: #G #E #B #N:#R:#T', 1);
		END_IF;
		step := 230;
	END_IF;

230:
	IF snd_step = 0 THEN
		snd_text := 'MIME-Version: 1.0';
		step := 250;
	END_IF;

250:
	IF snd_step = 0 THEN
		snd_text := 'Content-Type: multipart/mixed;boundary="x"';
		snd_lf_cnt := 2;
		step := 260;
	END_IF;

260:
	IF snd_step = 0 THEN
		snd_enable := TRUE;
		snd_text := 'This is a multi-part message in MIME format.';
		step := 270;
	END_IF;

270:
	IF snd_step = 0 THEN
		snd_enable := FALSE;
		snd_text := '--x';
		snd_lf_cnt := 1;
		step := 280;
	END_IF;

280:
	IF snd_step = 0 THEN
		snd_text := 'Content-Type: text/plain; format=flowed; charset="iso-8859-1";';
		snd_text := CONCAT(snd_text,' reply-type=original'); (* PCWORX kann nur konstanten mit max 80 zeichen *)
		step := 290;
	END_IF;

290:
	IF snd_step = 0 THEN
		snd_text := 'Content-Transfer-Encoding: 8bit';
		snd_lf_cnt := 2;
		step := 300;
	END_IF;

300:
	IF snd_step = 0 THEN
		snd_enable := TRUE;
		snd_text := BODY;
		snd_lf_cnt := 2;
		step := 310;
	END_IF;

310:
	IF snd_step = 0 THEN
		cnt1 := ELEMENT_COUNT(59, FILES) - 1; (* Anzahl der Dateien *)
		step := 400;
	END_IF;

(* +++++++++++++ File-Attachment ++++++++++++ *)
400:
	IF cnt1 >= 0 THEN
		str1 := ELEMENT_GET(59, cnt1, FILES);
		FILE_PATH_SPLIT(FILENAME:=str1,X:=fpd); (* Datei-Path zerlegen *)
		IF fpd.FILENAME = '#DEL#' THEN
			file_delete := TRUE;
		ELSE
			step := 410;
		END_IF;
		cnt1 := cnt1 - 1;
	ELSE
		step := 800;
	END_IF;

410:
	IF snd_step = 0 THEN
		snd_enable := FALSE;
		snd_text := '--x';
		snd_lf_cnt := 1;
		step := 420;
	END_IF;

420:
	IF snd_step = 0 THEN
		snd_text := 'Content-Transfer-Encoding: BASE64';
		str2 := CONCAT(fpd.FILENAME,'"');
		step := 430;
	END_IF;

430:
	IF snd_step = 0 THEN
		snd_text := CONCAT('Content-Type: application/octet-stream; name="',str2);
		step := 440;
	END_IF;

440:
	IF snd_step = 0 THEN
		snd_enable := TRUE;
		snd_text := CONCAT('Content-Disposition: attachment; filename="',str2);
		snd_lf_cnt := 2;
		step := 450;
	END_IF;

450:
	IF snd_step = 0 THEN
		FSD.FILENAME := str1; (* Dateiname *)
		FSD.OFFSET := UDINT#0; (* Start bei Dateianfang *)
		step := 460;
	END_IF;

460:
	FSD.MODE := BYTE#1; (* vorhandene Datei zum lesen öffnen *)
	F_BUF.SIZE := b64_max; (* maximale länge einlesen *)
	idx1 := 0;
	idx2 := 0;
	step := 470;

470:
	IF FSD.MODE = BYTE#0 AND FSD.ERROR = BYTE#0 THEN
		last_block := FSD.FILE_SIZE = FSD.OFFSET;
		b64_size1 := MIN(48,UINT_TO_INT(F_BUF.SIZE) - idx1);
		IF b64_size1 > 0 THEN
			idx3 := b64_size1 - 1;
			FOR i1 := 0 TO idx3 DO (* daten in BASE64 buffer kopieren *)
				b64_buf1[i1] := F_BUF.BUFFER[idx1];
				idx1 := idx1 + 1;
			END_FOR;
			BASE64_ENCODE_STREAM( SIZE1:= b64_size1, BUF1:= b64_buf1, BUF2:= b64_buf2, SIZE2=> b64_size2); (* BASE64 Kodierung *)
			idx3 := b64_size2 - 1;
			FOR i1 := 0 TO idx3 DO (* Daten aus BASE64 buffer kopieren *)
				S_BUF.BUFFER[idx2] := b64_buf2[i1];
				idx2 := idx2 + 1;
			END_FOR;
			b64_lf := TRUE;
			(*####################  DEBUG-MESSAGE  ###################################*)
			(*IF _debug_enable THEN
				LOG_CL.NEW_MSG := 'B64: FILE ~1 /SIZE ~2 /OFF ~3 /BSIZE ~4 /idx1 ~5 /idx2 ~6';
				LOG_CL.PRINTF[1] := FSD.FILENAME;
				LOG_CL.PRINTF[2] := UDINT_TO_STRING(FSD.FILE_SIZE);
				LOG_CL.PRINTF[3] := UDINT_TO_STRING(FSD.OFFSET);
				LOG_CL.PRINTF[4] := INT_TO_STRING(b64_size1);
				LOG_CL.PRINTF[5] := INT_TO_STRING(idx1);
				LOG_CL.PRINTF[6] := INT_TO_STRING(idx2);
				LOG_MSG();
			END_IF;*)
			(*########################################################################*)
		ELSE
			b64_lf := last_block;
			step := 480; (* block beendet  *)
		END_IF;
		IF b64_lf THEN
			S_BUF.BUFFER[idx2] := BYTE#16#0D;
			idx2 := idx2 + 1;
			S_BUF.BUFFER[idx2] := BYTE#16#0A;
			idx2 := idx2 + 1;
		END_IF;
		(*####################  DEBUG-MESSAGE  ###################################*)
		(*IF _debug_enable THEN
			LOG_CL.NEW_MSG := 'B64: exit ~1 /SIZE ~2 /OFF ~3 /eof ~4 /lf_cnt ~5';
			LOG_CL.PRINTF[1] := FSD.FILENAME;
			LOG_CL.PRINTF[2] := UDINT_TO_STRING(FSD.FILE_SIZE);
			LOG_CL.PRINTF[3] := UDINT_TO_STRING(FSD.OFFSET);
			LOG_CL.PRINTF[4] := BOOL_TO_STRING(last_block);
			LOG_CL.PRINTF[5] := INT_TO_STRING(snd_lf_cnt);
			LOG_MSG();
		END_IF;*)
		(*########################################################################*)
	END_IF;

480:
	S_BUF.SIZE := INT_TO_UINT(idx2); (* Daten senden *)
	(*####################  DEBUG-MESSAGE  ###################################*)
	(*IF _debug_enable THEN
		LOG_CL.NEW_MSG := 'B64: tcp_send ~1';
		LOG_CL.PRINTF[1] := INT_TO_STRING(idx2);
		LOG_MSG();
	END_IF;*)
	(*########################################################################*)
	step := 490;

490:
	IF S_BUF.SIZE = UINT#0 THEN (* warten bis alle daten gesendet sind *)
		step := SEL(last_block ,460,400);
	END_IF;

(* ++++++++++++++++++++++++++++++++++++++++ *)

800:
	IF snd_step = 0 THEN
		snd_enable := FALSE;
		snd_text := '--x--';
		snd_lf_cnt := 2;
		step := 810;
	END_IF;

810:
	IF snd_step = 0 THEN
		snd_enable := TRUE;
		snd_text := '.';
		snd_lf_cnt := 1;
		step := 820;
	END_IF;

820:
	IF rcv_state = 250 THEN (* 250 = Requested mail action okay *)
		snd_text := 'QUIT';
		ip_c_red_disable := TRUE;
		next_step := 830;
	END_IF;

830:
	IF rcv_state = 221  OR TON_WAIT.ET > timeout3 THEN (* 221 = Service closing transmission channel *)
		step := 900;
	END_IF;

(* ================================================== *)

900:
	IF FILE_DELETE THEN (* Dateien nach transfer löschen *)
		cnt1 := ELEMENT_COUNT(59, FILES) - 1; (* Trennzeichen >;< , Anzahl der Dateien *)
		step := 910;
	ELSE
		step := 950;
	END_IF;

910:
	IF FSD.MODE = BYTE#0 AND FSD.ERROR = BYTE#0 THEN
		IF cnt1 >= 0 THEN
			str1 := ELEMENT_GET(59, cnt1, FILES); (* Trennzeichen >;< *)
			IF str1 <> '#DEL#' THEN
				FSD.FILENAME := str1;
				FSD.MODE := BYTE#4; (* File Remove *)
			END_IF;
			cnt1 := cnt1 - 1;
		ELSE
			step := 950;
		END_IF;
	END_IF;

950:
	DONE := TRUE;
	step := 980;

980:
	IP_C.C_ENABLE := FALSE; (* SMTP Steuerkanal schliessen *)
	S_BUF.SIZE := UINT#0;
	R_BUF.SIZE := UINT#0;
	IP_C.MAILBOX[3] := BYTE#0; (* IP Empfang wieder freigeben *)
	snd_step := 0;
	next_step := 0;
	FSD.MODE := BYTE#5; (* Datei schliessen *)
	step := 990;

990:
	IF IP_C.C_STATE = BYTE#0 AND FSD.FILE_OPEN = FALSE THEN
		step := 0;
	END_IF;

(*  +++++++++++++++++ Authentifizierung +++++++++++++++++ *)

(* PLAIN ++++++++++++++++++++++++++++++++++++++++++++++++++++++++++ *)

1000:
	snd_text := CONCAT('AUTH',str3);
	snd_lf_cnt := 1;
 	step := 1010;

1010:
	IF rcv_state = 334 THEN (* 334 = Authentifizierung  *)
		cnt1 := LEN(URL_DATA.USER);
		cnt2 := LEN(URL_DATA.PASSWORD);
		IF cnt1 + cnt2 <= 46 THEN (* USER + PASSWORD dürfen zusammen maximal 46 Zeichen haben *)
			b64_buf1[0] := BYTE#0;
			FOR i1 := 1 TO cnt1 DO
				b64_buf1[i1] := OSCAT_BASIC.CODE(URL_DATA.USER, i1);
			END_FOR;
			b64_size1 := cnt1 + 1;
			b64_buf1[b64_size1] := BYTE#0;
			b64_size1 := b64_size1 + 1;
			FOR i1 := 1 TO cnt2 DO
				b64_buf1[b64_size1] := OSCAT_BASIC.CODE(URL_DATA.PASSWORD, i1);
				b64_size1 := b64_size1 + 1;
			END_FOR;
			BASE64_ENCODE_STREAM( SIZE1:= b64_size1, BUF1:= b64_buf1, BUF2:= b64_buf2, SIZE2=> b64_size2); (* BASE64 Kodierung *)
			idx1 := b64_size2 - 1;
			FOR i1 := 0 TO idx1 DO
				S_BUF.BUFFER[i1] := b64_buf2[i1];
			END_FOR;
			S_BUF.BUFFER[b64_size2] := BYTE#16#0D;
			b64_size2 := b64_size2 + 1;
			S_BUF.BUFFER[b64_size2] := BYTE#16#0A;
			b64_size2 := b64_size2 + 1;
			S_BUF.SIZE := INT_TO_UINT(b64_size2);
			rcv_state := 0;
		END_IF;
		step := 90;
	END_IF;

(* LOGIN ++++++++++++++++++++++++++++++++++++++++++++++++++++++++++ *)

1100:
	snd_text := CONCAT('AUTH',str3);
	snd_lf_cnt := 1;
 	step := 1110;

1110:
	IF rcv_state = 334 THEN (* 334 = Authentifizierung  *)
		b64_str1 := URL_DATA.USER;
		b64_start := TRUE; (* BASE64 kodierung von Username *)
		step := 1120;
	END_IF;

1120:
	IF b64_start AND b64_done THEN
		b64_start := FALSE;
		snd_text := b64_str2;
		next_step := 1130;
	END_IF;

1130:
	IF rcv_state = 334 THEN (* 334 = Password:  *)
		b64_str1 := URL_DATA.PASSWORD;
		b64_start := TRUE; (* BASE64 kodierung von Password *)
		step := 1140;
	END_IF;

1140:
	IF b64_start AND b64_done THEN
		b64_start := FALSE;
		snd_text := b64_str2;
		next_step := 90;
	END_IF;

(* CRAM-MD5  ++++++++++++++++++++++++++++++++++++++++++++++++++++++++++
(Challenge-Response Authentication Mechanism, Message Digest 5) Authentifizierung auf Basis von MD5-HMAC-Algorithmus. *)

1200:
	snd_text := CONCAT('AUTH',str3);
	snd_lf_cnt := 1;
 	step := 1210;

1210:
	IF rcv_state = 334 THEN (* 334 = Authentifizierung  *)
		md5_b64_ts := RIGHT(rcv_text,LEN(rcv_text) - 4);
		md5_user := URL_DATA.USER;
		md5_password := URL_DATA.PASSWORD;
		MD5_RUN := TRUE;
		step := 1220;
	END_IF;

1220:
	MD5_CRAM_AUTH(RUN:=MD5_RUN,USERNAME:=md5_user,PASSWORD:=md5_password,B64_TS:=md5_b64_ts,AUTH_KEY:=md5_auth_key);
	IF NOT MD5_RUN THEN
		snd_text := md5_auth_key;
		step := 90;
	END_IF;

(* STARTTLS  ++++++++++++++++++++++++++++++++++++++++++++++++++++++++++ *)

1300:
	snd_text := 'STARTTLS';
	snd_lf_cnt := 1;
 	step := 1310;

1310:
	IF rcv_state = 220 THEN (* 220 = Service ready - Ready to start TLS *)
		IP_C.MAILBOX[16] := BYTE#1; (* SSL/TLS aktivieren *)
		step := 1320;
	END_IF;

1320:
	IF IP_C.MAILBOX[16] = BYTE#2 THEN (* warten bis SSL/TLS aktiviert wurde *)
		step := 30; (* ganzer Ablauf von vorne beginnen *)
	END_IF;

(* keine Authentifizierung gefunden +++++++++++++++++++++++++++++++ *)
1900: ; (* Auf Laufzeitfehler warten *)

END_CASE;
(* ++++++++++++++++++++++++++++++++++++++++++++++++++++++++++ *)
IF step >= 30 THEN
	IF R_BUF.SIZE > UINT#0 THEN (* Daten wurden empfangen ? *)
		idx1 := UINT_TO_INT(R_BUF.SIZE);
		REPEAT (* zeilenterminierung erkennen und echtes TEXT-Ende bestimmen *)
			idx1 := idx1 - 1;
		UNTIL idx1 = 0 OR R_BUF.BUFFER[idx1] >= BYTE#32 (* TRUE = EXIT *)
		END_REPEAT;
		FOR i1 := 0 TO idx1 DO (* bei multiline alle CRLF durch >^< ersetzen *)
			IF R_BUF.BUFFER[i1] < BYTE#32 THEN
				R_BUF.BUFFER[i1] := BYTE#94; (* >^< *)
			END_IF;
		END_FOR;
		rcv_text := OSCAT_BASIC.BUFFER_TO_STRING(PT:=ADR(R_BUF.BUFFER),SIZE:=idx1+1,START:=0,STOP:=OSCAT_BASIC.STRING_LENGTH-1);
		IF LEN(rcv_text) >= 3 THEN (* Statuscode prüfen und auswerten *)
			rcv_s := LEFT(rcv_text,3);
			IF OSCAT_BASIC.IS_NUM(STR:=rcv_s) THEN (* enthält nur Zahlen ? *)
				rcv_state := STRING_TO_INT(rcv_s);
			END_IF;
			IP_C.R_OBSERVE := FALSE;
		END_IF;
		R_BUF.SIZE := UINT#0; (* daten löschen *)

		(*####################  DEBUG-MESSAGE  ###################################*)
		(*IF _debug_enable THEN
			LOG_CL.NEW_MSG := 'RCV: >~1<';
			LOG_CL.PRINTF[1] := rcv_text;
			LOG_MSG();
		END_IF;*)
		(*########################################################################*)

	END_IF;
END_IF;

(* automatisches Datensenden *)

CASE snd_step OF

00:
	IF LEN(snd_text) > 0 THEN

		(*####################  DEBUG-MESSAGE  ###################################*)
		(*IF _debug_enable THEN
			LOG_CL.NEW_MSG := 'SND: >~1< /lf ~2';
			LOG_CL.PRINTF[1] := snd_text;
			LOG_CL.PRINTF[2] := INT_TO_STRING(snd_lf_cnt);
			LOG_MSG();
		END_IF;*)
		(*########################################################################*)

		OSCAT_BASIC._STRING_TO_BUFFER(str:=snd_text,pos:=snd_idx,pt:=ADR(S_BUF.BUFFER),size:=SIZEOF(S_BUF.BUFFER)); (* String in puffer kopieren *)
		snd_idx := snd_idx + LEN(snd_text);
		FOR i1 := 1 TO snd_lf_cnt DO
			S_BUF.BUFFER[snd_idx] := BYTE#16#0D;
			snd_idx := snd_idx + 1;
			S_BUF.BUFFER[snd_idx] := BYTE#16#0A;
			snd_idx := snd_idx + 1;
		END_FOR;
		snd_text := '';
		rcv_state := 9999; (* letzen SMTP Status löschen *)

		IF snd_enable THEN
			S_BUF.SIZE := INT_TO_UINT(snd_idx); (* Sendelänge eintragen *)
			R_BUF.SIZE := UINT#0; (* Empfangsbuffer rücksetzen *)
			IP_C.R_OBSERVE := step <= 120 OR step >= 820;
			snd_idx := 0;
			snd_step := 10;
		END_IF;
	END_IF;

10:
	IF S_BUF.SIZE = UINT#0 THEN (* warten bis alle daten gesendet sind *)
		IF next_step <> 0 THEN
			step := next_step;
			next_step := 0;
		END_IF;
		snd_step := 0;
	END_IF;

END_CASE;

(* Globale Fehlerbehandlung für Haupt-Routine *)
IF ERROR_T = BYTE#0 AND step > 20 THEN (* noch kein Fehler gespeichert und Hauptroutine aktiv *)

	IF IP_C.ERROR > DWORD#0 AND IP_C.C_ENABLE AND NOT IP_C.TIME_RESET THEN  (* IP Control 1 *)
		IF ip_c_red_disable = FALSE OR IP_C.ERROR <> DWORD#16#FD000000 THEN
			ERROR_C := IP_C.ERROR;
			ERROR_T := BYTE#2;
			step := 980;
		END_IF;
	END_IF;

	IF FSD.MODE = BYTE#0 THEN
		IF FSD.ERROR > BYTE#0 THEN
			ERROR_C := BYTE_TO_DWORD(FSD.ERROR);
			ERROR_T := BYTE#4; (* Dateizugriff *)
			step := 980;
		END_IF;
	END_IF;
END_IF;

IF TON_WAIT.Q THEN (* Ablaufstörung - Schrittkette *)
	ERROR_C := SHL(INT_TO_DWORD(step),16) OR INT_TO_DWORD(rcv_state); (* aktuellen Schritt und letzten SMTP Status eintragen *)
	ERROR_T := BYTE#5;
	step := 980;
END_IF;

